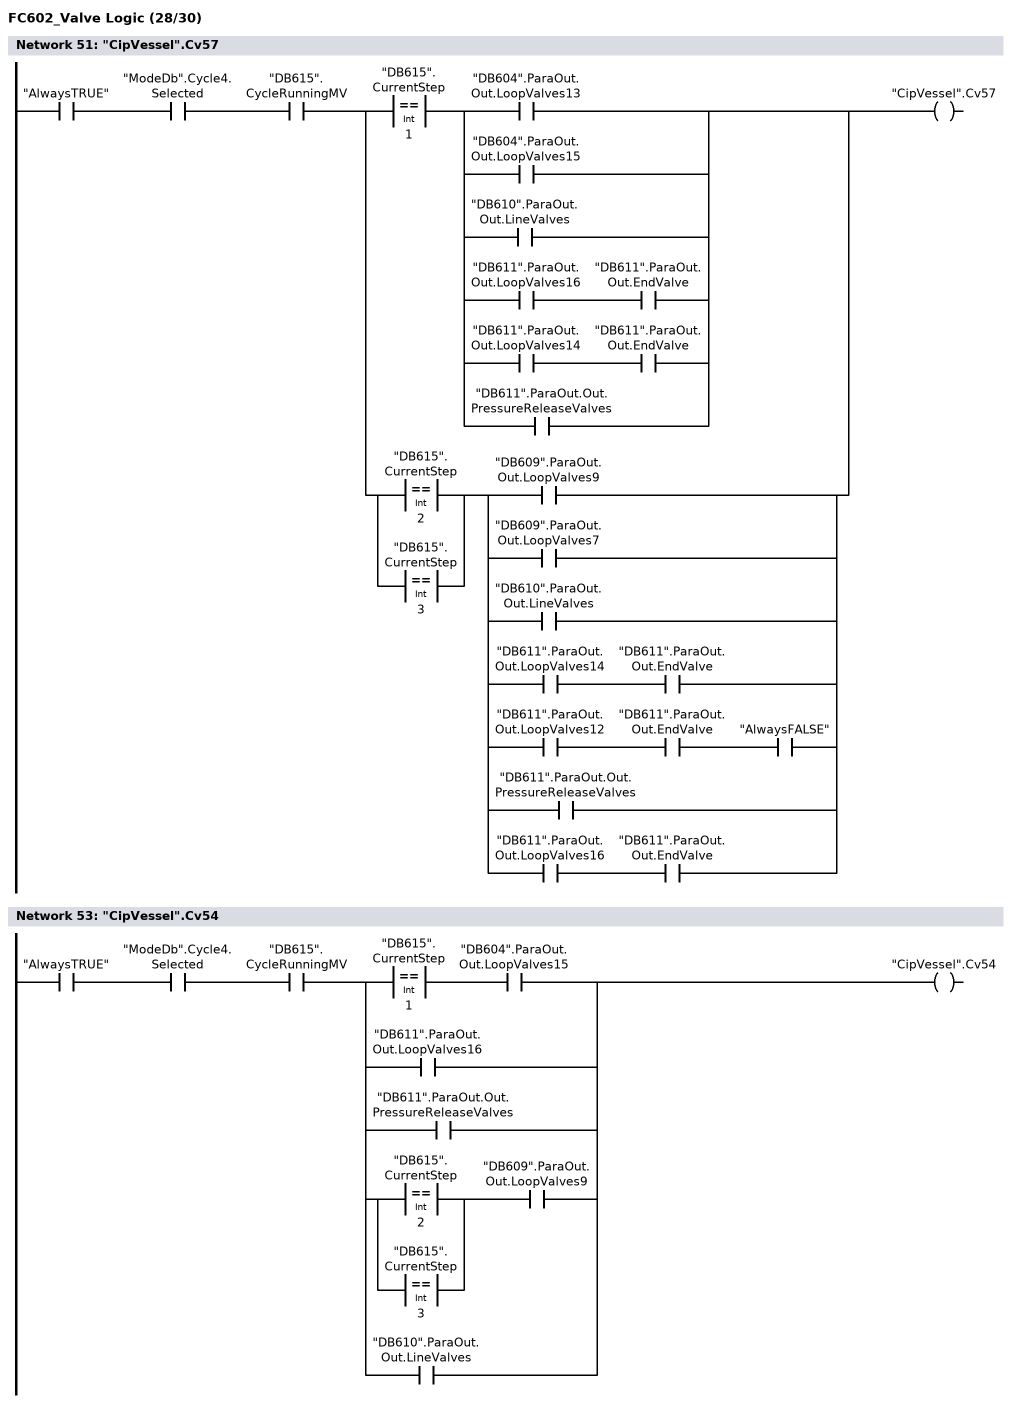
   RUNG wire#powerrail
      Contact( "AlwaysTRUE" )
      Contact( "ModeDb".Cycle4.Selected )
      Contact( "DB615".CycleRunningMV )
      wire#w1
      { S7_Templates := "SrcType := Int" } EQ_Contact(in1 := "DB615".CurrentStep, in2 := 1)
      wire#w2
      Contact( "DB604".ParaOut.Out.LoopValves13 )
      wire#w3
      Coil( "CipVessel".Cv57 )
   END_RUNG
   RUNG wire#w2
      Contact( "DB604".ParaOut.Out.LoopValves15 )
   END_RUNG wire#w3
   RUNG wire#w2
      Contact( "DB610".ParaOut.Out.LineValves )
   END_RUNG wire#w3
   RUNG wire#w2
      Contact( "DB611".ParaOut.Out.LoopValves16 )
      Contact( "DB611".ParaOut.Out.EndValve )
   END_RUNG wire#w3
   RUNG wire#w2
      Contact( "DB611".ParaOut.Out.LoopValves14 )
      Contact( "DB611".ParaOut.Out.EndValve )
   END_RUNG wire#w3
   RUNG wire#w2
      Contact( "DB611".ParaOut.Out.PressureReleaseValves )
   END_RUNG wire#w3
   RUNG wire#w1
      { S7_Templates := "SrcType := Int" } EQ_Contact(in1 := "DB615".CurrentStep, in2 := 2)
      wire#w4
      Contact( "DB609".ParaOut.Out.LoopValves9 )
   END_RUNG wire#w3
   RUNG wire#w1
      { S7_Templates := "SrcType := Int" } EQ_Contact(in1 := "DB615".CurrentStep, in2 := 3)
   END_RUNG wire#w4
   RUNG wire#w4
      Contact( "DB609".ParaOut.Out.LoopValves7 )
   END_RUNG wire#w3
   RUNG wire#w4
      Contact( "DB610".ParaOut.Out.LineValves )
   END_RUNG wire#w3
   RUNG wire#w4
      Contact( "DB611".ParaOut.Out.LoopValves14 )
      Contact( "DB611".ParaOut.Out.EndValve )
   END_RUNG wire#w3
   RUNG wire#w4
      Contact( "DB611".ParaOut.Out.LoopValves12 )
      Contact( "DB611".ParaOut.Out.EndValve )
      Contact( "AlwaysFALSE" )
   END_RUNG wire#w3
   RUNG wire#w4
      Contact( "DB611".ParaOut.Out.PressureReleaseValves )
   END_RUNG wire#w3
   RUNG wire#w4
      Contact( "DB611".ParaOut.Out.LoopValves16 )
      Contact( "DB611".ParaOut.Out.EndValve )
   END_RUNG wire#w3
   // the same network as SCL:
   "CipVessel".Cv57 := "AlwaysTRUE" AND "ModeDb".Cycle4.Selected AND "DB615".CycleRunningMV AND ((("DB615".CurrentStep = 1) AND ("DB604".ParaOut.Out.LoopValves13 OR "DB604".ParaOut.Out.LoopValves15 OR "DB610".ParaOut.Out.LineValves OR ("DB611".ParaOut.Out.LoopValves16 AND "DB611".ParaOut.Out.EndValve) OR ("DB611".ParaOut.Out.LoopValves14 AND "DB611".ParaOut.Out.EndValve) OR "DB611".ParaOut.Out.PressureReleaseValves)) OR ((("DB615".CurrentStep = 2) OR ("DB615".CurrentStep = 3)) AND ("DB609".ParaOut.Out.LoopValves9 OR "DB609".ParaOut.Out.LoopValves7 OR "DB610".ParaOut.Out.LineValves OR ("DB611".ParaOut.Out.LoopValves14 AND "DB611".ParaOut.Out.EndValve) OR ("DB611".ParaOut.Out.LoopValves12 AND "DB611".ParaOut.Out.EndValve AND "AlwaysFALSE") OR "DB611".ParaOut.Out.PressureReleaseValves OR ("DB611".ParaOut.Out.LoopValves16 AND "DB611".ParaOut.Out.EndValve))));
END_REGION

REGION Network 52: ---------- PTL LINE ------------
END_REGION

REGION Network 53: "CipVessel".Cv54
   RUNG wire#powerrail
      Contact( "AlwaysTRUE" )
      Contact( "ModeDb".Cycle4.Selected )
      Contact( "DB615".CycleRunningMV )
      wire#w1
      { S7_Templates := "SrcType := Int" } EQ_Contact(in1 := "DB615".CurrentStep, in2 := 1)
      Contact( "DB604".ParaOut.Out.LoopValves15 )
      wire#w2
      Coil( "CipVessel".Cv54 )
   END_RUNG
   RUNG wire#w1
      Contact( "DB611".ParaOut.Out.LoopValves16 )
   END_RUNG wire#w2
   RUNG wire#w1
      Contact( "DB611".ParaOut.Out.PressureReleaseValves )
   END_RUNG wire#w2
   RUNG wire#w1
      { S7_Templates := "SrcType := Int" } EQ_Contact(in1 := "DB615".CurrentStep, in2 := 2)
      wire#w3
      Contact( "DB609".ParaOut.Out.LoopValves9 )
   END_RUNG wire#w2
   RUNG wire#w1
      { S7_Templates := "SrcType := Int" } EQ_Contact(in1 := "DB615".CurrentStep, in2 := 3)
   END_RUNG wire#w3
   RUNG wire#w1
      Contact( "DB610".ParaOut.Out.LineValves )
   END_RUNG wire#w2
   // the same network as SCL:
   "CipVessel".Cv54 := "AlwaysTRUE" AND "ModeDb".Cycle4.Selected AND "DB615".CycleRunningMV AND ((("DB615".CurrentStep = 1) AND "DB604".ParaOut.Out.LoopValves15) OR "DB611".ParaOut.Out.LoopValves16 OR "DB611".ParaOut.Out.PressureReleaseValves OR ((("DB615".CurrentStep = 2) OR ("DB615".CurrentStep = 3)) AND "DB609".ParaOut.Out.LoopValves9) OR "DB610".ParaOut.Out.LineValves);
END_REGION

REGION Network 54: "CipVessel".Cv55
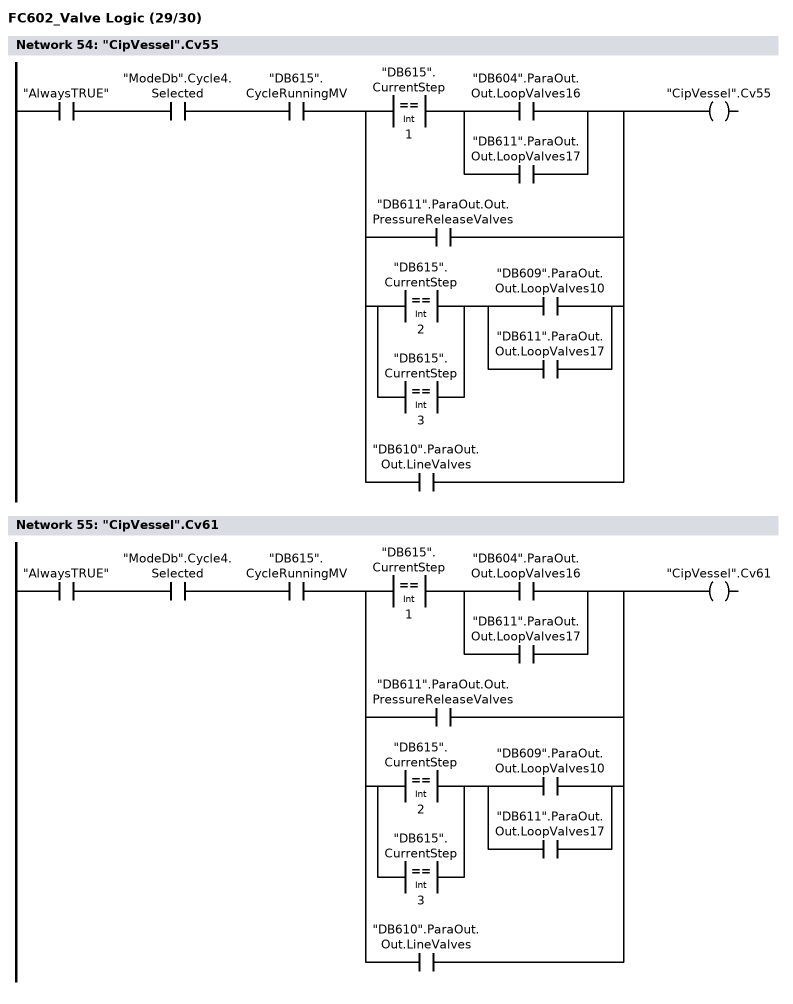
   RUNG wire#powerrail
      Contact( "AlwaysTRUE" )
      Contact( "ModeDb".Cycle4.Selected )
      Contact( "DB615".CycleRunningMV )
      wire#w1
      { S7_Templates := "SrcType := Int" } EQ_Contact(in1 := "DB615".CurrentStep, in2 := 1)
      wire#w2
      Contact( "DB604".ParaOut.Out.LoopValves16 )
      wire#w3
      Coil( "CipVessel".Cv55 )
   END_RUNG
   RUNG wire#w2
      Contact( "DB611".ParaOut.Out.LoopValves17 )
   END_RUNG wire#w3
   RUNG wire#w1
      Contact( "DB611".ParaOut.Out.PressureReleaseValves )
   END_RUNG wire#w3
   RUNG wire#w1
      { S7_Templates := "SrcType := Int" } EQ_Contact(in1 := "DB615".CurrentStep, in2 := 2)
      wire#w4
      Contact( "DB609".ParaOut.Out.LoopValves10 )
   END_RUNG wire#w3
   RUNG wire#w1
      { S7_Templates := "SrcType := Int" } EQ_Contact(in1 := "DB615".CurrentStep, in2 := 3)
   END_RUNG wire#w4
   RUNG wire#w4
      Contact( "DB611".ParaOut.Out.LoopValves17 )
   END_RUNG wire#w3
   RUNG wire#w1
      Contact( "DB610".ParaOut.Out.LineValves )
   END_RUNG wire#w3
   // the same network as SCL:
   "CipVessel".Cv55 := "AlwaysTRUE" AND "ModeDb".Cycle4.Selected AND "DB615".CycleRunningMV AND ((("DB615".CurrentStep = 1) AND ("DB604".ParaOut.Out.LoopValves16 OR "DB611".ParaOut.Out.LoopValves17)) OR "DB611".ParaOut.Out.PressureReleaseValves OR ((("DB615".CurrentStep = 2) OR ("DB615".CurrentStep = 3)) AND ("DB609".ParaOut.Out.LoopValves10 OR "DB611".ParaOut.Out.LoopValves17)) OR "DB610".ParaOut.Out.LineValves);
END_REGION

REGION Network 55: "CipVessel".Cv61
   RUNG wire#powerrail
      Contact( "AlwaysTRUE" )
      Contact( "ModeDb".Cycle4.Selected )
      Contact( "DB615".CycleRunningMV )
      wire#w1
      { S7_Templates := "SrcType := Int" } EQ_Contact(in1 := "DB615".CurrentStep, in2 := 1)
      wire#w2
      Contact( "DB604".ParaOut.Out.LoopValves16 )
      wire#w3
      Coil( "CipVessel".Cv61 )
   END_RUNG
   RUNG wire#w2
      Contact( "DB611".ParaOut.Out.LoopValves17 )
   END_RUNG wire#w3
   RUNG wire#w1
      Contact( "DB611".ParaOut.Out.PressureReleaseValves )
   END_RUNG wire#w3
   RUNG wire#w1
      { S7_Templates := "SrcType := Int" } EQ_Contact(in1 := "DB615".CurrentStep, in2 := 2)
      wire#w4
      Contact( "DB609".ParaOut.Out.LoopValves10 )
   END_RUNG wire#w3
   RUNG wire#w1
      { S7_Templates := "SrcType := Int" } EQ_Contact(in1 := "DB615".CurrentStep, in2 := 3)
   END_RUNG wire#w4
   RUNG wire#w4
      Contact( "DB611".ParaOut.Out.LoopValves17 )
   END_RUNG wire#w3
   RUNG wire#w1
      Contact( "DB610".ParaOut.Out.LineValves )
   END_RUNG wire#w3
   // the same network as SCL:
   "CipVessel".Cv61 := "AlwaysTRUE" AND "ModeDb".Cycle4.Selected AND "DB615".CycleRunningMV AND ((("DB615".CurrentStep = 1) AND ("DB604".ParaOut.Out.LoopValves16 OR "DB611".ParaOut.Out.LoopValves17)) OR "DB611".ParaOut.Out.PressureReleaseValves OR ((("DB615".CurrentStep = 2) OR ("DB615".CurrentStep = 3)) AND ("DB609".ParaOut.Out.LoopValves10 OR "DB611".ParaOut.Out.LoopValves17)) OR "DB610".ParaOut.Out.LineValves);
END_REGION

REGION Network 56: "CipVessel".Cv60
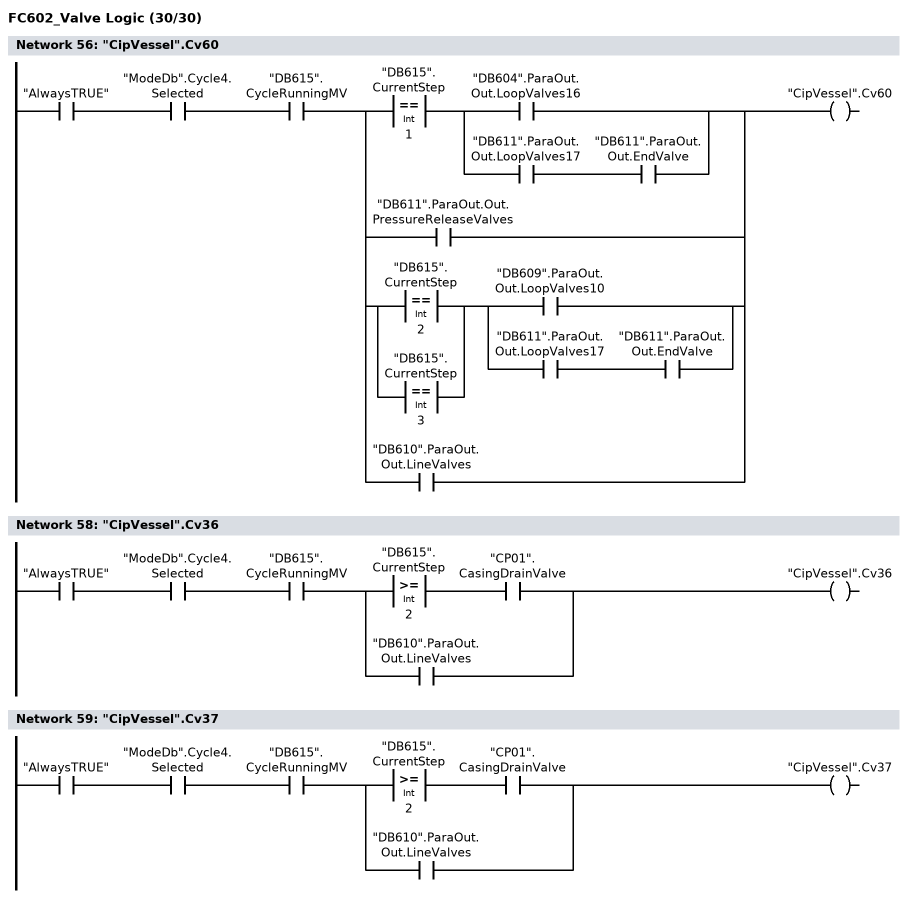
   RUNG wire#powerrail
      Contact( "AlwaysTRUE" )
      Contact( "ModeDb".Cycle4.Selected )
      Contact( "DB615".CycleRunningMV )
      wire#w1
      { S7_Templates := "SrcType := Int" } EQ_Contact(in1 := "DB615".CurrentStep, in2 := 1)
      wire#w2
      Contact( "DB604".ParaOut.Out.LoopValves16 )
      wire#w3
      Coil( "CipVessel".Cv60 )
   END_RUNG
   RUNG wire#w2
      Contact( "DB611".ParaOut.Out.LoopValves17 )
      Contact( "DB611".ParaOut.Out.EndValve )
   END_RUNG wire#w3
   RUNG wire#w1
      Contact( "DB611".ParaOut.Out.PressureReleaseValves )
   END_RUNG wire#w3
   RUNG wire#w1
      { S7_Templates := "SrcType := Int" } EQ_Contact(in1 := "DB615".CurrentStep, in2 := 2)
      wire#w4
      Contact( "DB609".ParaOut.Out.LoopValves10 )
   END_RUNG wire#w3
   RUNG wire#w1
      { S7_Templates := "SrcType := Int" } EQ_Contact(in1 := "DB615".CurrentStep, in2 := 3)
   END_RUNG wire#w4
   RUNG wire#w4
      Contact( "DB611".ParaOut.Out.LoopValves17 )
      Contact( "DB611".ParaOut.Out.EndValve )
   END_RUNG wire#w3
   RUNG wire#w1
      Contact( "DB610".ParaOut.Out.LineValves )
   END_RUNG wire#w3
   // the same network as SCL:
   "CipVessel".Cv60 := "AlwaysTRUE" AND "ModeDb".Cycle4.Selected AND "DB615".CycleRunningMV AND ((("DB615".CurrentStep = 1) AND ("DB604".ParaOut.Out.LoopValves16 OR ("DB611".ParaOut.Out.LoopValves17 AND "DB611".ParaOut.Out.EndValve))) OR "DB611".ParaOut.Out.PressureReleaseValves OR ((("DB615".CurrentStep = 2) OR ("DB615".CurrentStep = 3)) AND ("DB609".ParaOut.Out.LoopValves10 OR ("DB611".ParaOut.Out.LoopValves17 AND "DB611".ParaOut.Out.EndValve))) OR "DB610".ParaOut.Out.LineValves);
END_REGION

REGION Network 57: ----------PCD DRAIN------------
END_REGION

REGION Network 58: "CipVessel".Cv36
   RUNG wire#powerrail
      Contact( "AlwaysTRUE" )
      Contact( "ModeDb".Cycle4.Selected )
      Contact( "DB615".CycleRunningMV )
      wire#w1
      { S7_Templates := "SrcType := Int" } GE_Contact(in1 := "DB615".CurrentStep, in2 := 2)
      Contact( "CP01".CasingDrainValve )
      wire#w2
      Coil( "CipVessel".Cv36 )
   END_RUNG
   RUNG wire#w1
      Contact( "DB610".ParaOut.Out.LineValves )
   END_RUNG wire#w2
   // the same network as SCL:
   "CipVessel".Cv36 := "AlwaysTRUE" AND "ModeDb".Cycle4.Selected AND "DB615".CycleRunningMV AND ((("DB615".CurrentStep >= 2) AND "CP01".CasingDrainValve) OR "DB610".ParaOut.Out.LineValves);
END_REGION

REGION Network 59: "CipVessel".Cv37
   RUNG wire#powerrail
      Contact( "AlwaysTRUE" )
      Contact( "ModeDb".Cycle4.Selected )
      Contact( "DB615".CycleRunningMV )
      wire#w1
      { S7_Templates := "SrcType := Int" } GE_Contact(in1 := "DB615".CurrentStep, in2 := 2)
      Contact( "CP01".CasingDrainValve )
      wire#w2
      Coil( "CipVessel".Cv37 )
   END_RUNG
   RUNG wire#w1
      Contact( "DB610".ParaOut.Out.LineValves )
   END_RUNG wire#w2
   // the same network as SCL:
   "CipVessel".Cv37 := "AlwaysTRUE" AND "ModeDb".Cycle4.Selected AND "DB615".CycleRunningMV AND ((("DB615".CurrentStep >= 2) AND "CP01".CasingDrainValve) OR "DB610".ParaOut.Out.LineValves);
END_REGION
END_FUNCTION

FUNCTION "FC615" : Void
{ S7_Optimized_Access := 'TRUE' }
VERSION : 0.1

BEGIN
	REGION Common
	    IF "DB615".SelectStep = TRUE THEN
	        "DB615".TempStep := "DB615".CurrentStep;
	        REPEAT
	        "DB615".TempStep := "DB615".TempStep + 1;
	        UNTIL "DB623".StepEnable["DB615".TempStep] = TRUE OR ("DB615".TempStep > "DB616".TotalStep) END_REPEAT;
	        IF "DB615".TempStep <= "DB616".TotalStep THEN
	            "DB615".CurrentStep := "DB615".TempStep;
	        ELSE
	            "DB615".ProcessOver := 1;
	        END_IF;         
	        "DB615".SelectStep := false;
	    END_IF;
	    
	    
	    
	    IF "DB622".MainPopupMsg2 = 1 THEN
	        POKE_BLK(area_src := 16#84,
	                 dbNumber_src := 626,
	                 byteOffset_src := 0,
	                 area_dest := 16#84,
	                 dbNumber_dest := 625,
	                 byteOffset_dest := 0,
	                 count := 2382);  
	    END_IF;
	    
	END_REGION
	
	REGION common Set Para
	    "DB603".CycleSelection := "DB616".CycleSelection["DB615".CurrentStep];
	    
	    "DB604".ParaIn := "DB616".FillingInputPara["DB615".CurrentStep];
	    "DB607".SetTimeSecs := "DB616".MixingTimeInput["DB615".CurrentStep];
	    "DB608".ParaIn := "DB616".RecirculationInput["DB615".CurrentStep];
	    "DB609".ParaIn := "DB616".DrainInputs["DB615".CurrentStep];
	    "DB610".SetTime := "DB616".SystemDrainSetTimeInput["DB615".CurrentStep];
	    "DB611".ParaIn := "DB616".AirPurgingInputPara["DB615".CurrentStep];
	    "DB603".CycleSelection := "DB616".CycleSelection["DB615".CurrentStep];
	    
	    "DB609".ActualPressure := "AiDb".Ai11.ActValue;
	    "DB627".RepSv := "DB616".CycleSelection["DB615".CurrentStep].StepSelection.SetRepetition;
	    "DB627".RepPv := "DB603".ActualRepetition;
	    "DB604".ActualQuantity := "ModeDb".VesselWeight;
	    "DB609".ActualWeight := "ModeDb".VesselWeight;
	  //  "DB611".ActualPressure := "AiDb".Ai07.ActValue;
	    "DB609".ActualConductivityVessel := "AiDb".Ai15.ActValue;
	    "DB609".ParaIn.Parameters.SetConductivity := "DB623".FinalRinseSetCond;
	    "DB611".ActualPressure := "DB615".ApActPressure;
	    
	
	    "DB616".DrainInputs["DB615".CurrentStep].PreciseEngineering.DrainWeight := "DB624".VesselDrainWeight;
	    "DB616".DrainInputs["DB615".CurrentStep].Parameters.SetPressure := "DB623".DrainPressure;
	    "DB616".DrainInputs["DB615".CurrentStep].Parameters.PressureTolerance := "DB624".DrainPressureTolerance;
	    "DB616".DrainInputs["DB615".CurrentStep].ProductionSetting.CaiDelay := "CommonProductionSettings".CAIDelay;
	    
	    "DB616".SystemDrainSetTimeInput["DB615".CurrentStep] := "DB623".SystemDrainTime;
	    
	    "DB616".AirPurgingInputPara["DB615".CurrentStep].Parameters.SetPressure := "DB623".AirPurgingPressure;
	    "DB616".AirPurgingInputPara["DB615".CurrentStep].Parameters.PressureTolerance := "DB624".AirPurgingPressureTolerence;
	    "DB616".AirPurgingInputPara["DB615".CurrentStep].Parameters.VentOnTime := "DB624".AirPurgingReleaseTime;
	    "DB616".AirPurgingInputPara["DB615".CurrentStep].ProductionSetting.CAIDelay := "CommonProductionSettings".CAIDelay;
	    
	    
	    IF "DB611".StepDelay."Noof StepsPv" <= 1 THEN
	        "DB616".AirPurgingInputPara["DB615".CurrentStep].Selections.PressureMode := 0;
	    ELSE
	        "DB616".AirPurgingInputPara["DB615".CurrentStep].Selections.PressureMode := 1;
	    END_IF;
	    
	    "DB616".AirPurgingInputPara["DB615".CurrentStep].ProductionSetting.LoopDelay1 := "DB624".AirPurgeSamplingLineDelay;
	    "DB616".AirPurgingInputPara["DB615".CurrentStep].ProductionSetting.LoopDelay2 := "DB624".AirPurgeBlankeingLineDelay;
	    "DB616".AirPurgingInputPara["DB615".CurrentStep].ProductionSetting.LoopDelay3 := "DB624".AirPurgeJTubeLineDelay;
	    "DB616".AirPurgingInputPara["DB615".CurrentStep].ProductionSetting.LoopDelay4 := "DB624".AirPurgeSpargingLineDelay;
	    "DB616".AirPurgingInputPara["DB615".CurrentStep].ProductionSetting.LoopDelay5 := "DB624".AirPurgeSbiLineDelay;
	    "DB616".AirPurgingInputPara["DB615".CurrentStep].ProductionSetting.LoopDelay6 := "DB624".AirPurgeRecirculationlineDelay;
	    "DB616".AirPurgingInputPara["DB615".CurrentStep].ProductionSetting.LoopDelay7 := "DB624".AirPurgeVesselBypassLineDelay;
	    "DB616".AirPurgingInputPara["DB615".CurrentStep].ProductionSetting.LoopDelay8 := "DB624".AirPurgeVesselDrainLineDelay;
	    "DB616".AirPurgingInputPara["DB615".CurrentStep].ProductionSetting.LoopDelay9 := "DB624".AirPurgePumpBypassLineDelay;
	    "DB616".AirPurgingInputPara["DB615".CurrentStep].ProductionSetting.LoopDelay10 := "DB624".AirPurgePf01InLineDelay;
	    "DB616".AirPurgingInputPara["DB615".CurrentStep].ProductionSetting.LoopDelay11 := "DB624".AirPurgePf01VentLineDelay;
	    "DB616".AirPurgingInputPara["DB615".CurrentStep].ProductionSetting.LoopDelay12 := "DB624".AirPurgePf02InLineDelay;
	    "DB616".AirPurgingInputPara["DB615".CurrentStep].ProductionSetting.LoopDelay13 := "DB624".AirPurgePf02VentLineDelay;
	    "DB616".AirPurgingInputPara["DB615".CurrentStep].ProductionSetting.LoopDelay14 := "DB624".AirPurgePf02OutLineDelay;
	    "DB616".AirPurgingInputPara["DB615".CurrentStep].ProductionSetting.LoopDelay15 := "DB624".AirPurgePf01BypassLineDelay;
	    "DB616".AirPurgingInputPara["DB615".CurrentStep].ProductionSetting.LoopDelay16 := "DB624".AirPurgePf02BypassLineDelay;
	    "DB616".AirPurgingInputPara["DB615".CurrentStep].ProductionSetting.LoopDelay17 := "DB624".AirPurgePtlLineDelay;
	    
	END_REGION
	
	REGION Cycle 1 - PRE RINSE  CYCLE
	    
	    "DB616".CycleSelection[1].StepSelection.SetRepetition := "DB623".PreRinseCycleNoOfRep;
	    
	    "DB616".FillingInputPara[1].ProductionSetting.ZDVDelay := "CommonProductionSettings".WFIDelay;
	    "DB616".FillingInputPara[1].Parameters.PulsingOnTime := "DB623".SbiOnTime;
	    "DB616".FillingInputPara[1].Parameters.PulsingOffTime := "DB623".SbiOffTime;
	
	    "DB616".FillingInputPara[1].ProductionSetting.LoopDelay1 := "DB624".FillRinseSamplingLineDelay;
	    "DB616".FillingInputPara[1].ProductionSetting.LoopDelay2 := "DB624".FillRinseBlanketingLineDelay;
	    "DB616".FillingInputPara[1].ProductionSetting.LoopDelay3 := "DB624".FillRinseJTubeLineDelay;
	    "DB616".FillingInputPara[1].ProductionSetting.LoopDelay4 := "DB624".FillRinseSpargingLineDelay;
	    "DB616".FillingInputPara[1].ProductionSetting.LoopDelay5 := "DB624".FillRinseSbiLineDelay;
	    "DB616".FillingInputPara[1].ProductionSetting.LoopDelay6 := "DB624".FillRinseRecirculationlineDelay;
	    "DB616".FillingInputPara[1].ProductionSetting.LoopDelay7 := "DB624".FillRinseVesselBypassLineDelay;
	    "DB616".FillingInputPara[1].ProductionSetting.LoopDelay8 := "DB624".FillRinsePumpBypassLineDelay;
	    "DB616".FillingInputPara[1].ProductionSetting.LoopDelay9 := "DB624".FillRinsePf01InLineDelay;
	    "DB616".FillingInputPara[1].ProductionSetting.LoopDelay10 := "DB624".FillRinsePf01VentLineDelay;
	    "DB616".FillingInputPara[1].ProductionSetting.LoopDelay11 := "DB624".FillRinsePf02InLineDelay;
	    "DB616".FillingInputPara[1].ProductionSetting.LoopDelay12 := "DB624".FillRinsePf02VentLineDelay;
	    "DB616".FillingInputPara[1].ProductionSetting.LoopDelay13 := "DB624".FillRinsePf02OutLineDelay;
	    "DB616".FillingInputPara[1].ProductionSetting.LoopDelay14 := "DB624".FillRinsePf01BypassLineDelay;
	    "DB616".FillingInputPara[1].ProductionSetting.LoopDelay15 := "DB624".FillRinsePf02BypassLineDelay;
	    "DB616".FillingInputPara[1].ProductionSetting.LoopDelay16 := "DB624".FillRinsePtlLineDelay;
	    
	    
	    // "DB616".AirPurgingInputPara[1].ProductionSetting.LoopDelay1 := "DB624".AirPurgeSamplingLineDelay;
	    // "DB616".AirPurgingInputPara[1].ProductionSetting.LoopDelay2 := "DB624".AirPurgeBlankeingLineDelay;
	    // "DB616".AirPurgingInputPara[1].ProductionSetting.LoopDelay3 := "DB624".AirPurgeJTubeLineDelay;
	    // "DB616".AirPurgingInputPara[1].ProductionSetting.LoopDelay4 := "DB624".AirPurgeSpargingLineDelay;
	    // "DB616".AirPurgingInputPara[1].ProductionSetting.LoopDelay5 := "DB624".AirPurgeSbiLineDelay;
	    // "DB616".AirPurgingInputPara[1].ProductionSetting.LoopDelay6 := "DB624".AirPurgeRecirculationlineDelay;
	    // "DB616".AirPurgingInputPara[1].ProductionSetting.LoopDelay7 := "DB624".AirPurgeVesselBypassLineDelay;
	    // "DB616".AirPurgingInputPara[1].ProductionSetting.LoopDelay8 := "DB624".AirPurgeVesselDrainLineDelay ;
	    // "DB616".AirPurgingInputPara[1].ProductionSetting.LoopDelay9 := "DB624".AirPurgePumpBypassLineDelay ;
	    // "DB616".AirPurgingInputPara[1].ProductionSetting.LoopDelay10 := "DB624".AirPurgePf01InLineDelay ;
	    // "DB616".AirPurgingInputPara[1].ProductionSetting.LoopDelay11 := "DB624".AirPurgePf01VentLineDelay ;
	    // "DB616".AirPurgingInputPara[1].ProductionSetting.LoopDelay12 := "DB624".AirPurgePf02InLineDelay ;
	    // "DB616".AirPurgingInputPara[1].ProductionSetting.LoopDelay13 := "DB624".AirPurgePf02VentLineDelay ;
	    // "DB616".AirPurgingInputPara[1].ProductionSetting.LoopDelay14 := "DB624".AirPurgePf02OutLineDelay ;
	    // "DB616".AirPurgingInputPara[1].ProductionSetting.LoopDelay15 := "DB624".AirPurgePf01BypassLineDelay ;
	    // "DB616".AirPurgingInputPara[1].ProductionSetting.LoopDelay16 := "DB624".AirPurgePf02BypassLineDelay ;
	    // "DB616".AirPurgingInputPara[1].ProductionSetting.LoopDelay17 :="DB624".AirPurgePtlLineDelay ;
	    
	    // CASE "DB611".StepDelay."Noof StepsPv" OF
	    //     0..5:
	    //         "DB616".AirPurgingInputPara[1].Selections.PressureMode := 1;
	    //     6:
	    //         "DB616".AirPurgingInputPara[1].Selections.PressureMode := 0;
	    //     7..16:
	    //         "DB616".AirPurgingInputPara[1].Selections.PressureMode := 1;
	    //     ELSE
	    //         "DB616".AirPurgingInputPara[1].Selections.PressureMode := 1;
	    // END_CASE;
	            
	    
	    
	    REGION FILLING
	        IF "DB615".CurrentStep = 1 THEN
	            "DB616".FillingOutputPara[1] := "DB604".ParaOut;
	            "DB625".FillingPrint[1] := "DB604".Print;
	        ELSE
	            "DB616".FillingOutputPara[1] := "DB616".FillingOutputPara[0];
	        END_IF;
	    END_REGION
	    
	    REGION DRAIN
	        IF "DB615".CurrentStep = 1 AND "DB609".CycleEnable = 1 THEN
	            "DB616".DrainOutputs[1] := "DB609".ParaOut;
	
	        ELSE
	            "DB616".DrainOutputs[2] := "DB616".DrainOutputs[0];
	        END_IF;
	    END_REGION
	    
	    REGION SYSTEM DRAIN      
	        IF "DB615".CurrentStep = 1 THEN
	            "DB616".SystemDrainOutPara[1] := "DB610".ParaOut;
	        ELSE
	            "DB616".SystemDrainOutPara[1] := "DB616".SystemDrainOutPara[0];
	        END_IF;
	    END_REGION
	    
	    REGION AIR PURGE
	        IF "DB615".CurrentStep = 1 THEN
	            "DB616".AirPurgingOutPara[1] := "DB611".ParaOut;
	        ELSE
	            "DB616".AirPurgingOutPara[1] := "DB616".AirPurgingOutPara[0];
	        END_IF;
	    END_REGION
	    
	    REGION ON SCREEN PV
	        IF "DB615".CurrentStep = 1 THEN
	            //"DB627".FillQtySv := "DB623".Cyc1FillQty;
	            "DB627".FillQtyPv := "DB604".ActualQuantity;
	            //"DB627".TempSv := "DB623".Cyc1SetTemp;
	           // "DB627".TempPv := "DB605".ActualTemperature;
	            "DB627".MixingPv := "DB607".MixingTimer.TimeSecPV;
	            "DB627".MixingSv := "DB616".MixingTimeInput[1];
	        //    "DB627".APSv := "DB616".AirPurgingOutPara[1].Out.TimeSV;
	            "DB627".ApPv := "DB616".AirPurgingOutPara[1].Out.TimePV;
	            "DB627".APSv := "DB611".ParaOut.Out.TimeSV;
	            "DB627".ApReleaseTimeSv := "DB616".AirPurgingInputPara[1].Parameters.VentOnTime;
	            "DB627".ApReleaseTimePv := "DB616".AirPurgingOutPara[1].Out.PressureReleaseTimePV;
	            "DB627".SdSv := "DB623".SystemDrainTime;
	            "DB627".SdPv := "DB610".TimePv;
	           "DB627".RecirculationSv := "DB616".RecirculationOutput[1].Out.TimeSV;
	           "DB627".RecirculationPv := "DB616".RecirculationOutput[1].Out.TimePV;
	           "DB627".ConductivitySv := "DB609".ParaIn.Parameters.SetConductivity;
	           "DB627".ConductivityPv := "DB609".ActualConductivityVessel;
	         //   "DB627".DosingTimeSv := 0;
	         //   "DB627".DosingTimePv := 0;
	            "DB627".ApSetPressureSv := "DB623".AirPurgingPressure;
	            "DB627".ApSetPressurePv := "DB611".ActualPressure;
	            
	        END_IF;
	    END_REGION
	END_REGION
	
	REGION Cycle 2 - FILLING CYCLE
	    
	    "DB616".CycleSelection[2].StepSelection.SetRepetition := "DB623".FillingCycleNoOfRep;
	    
	    "DB616".FillingInputPara[2].ProductionSetting.ZDVDelay := "CommonProductionSettings".WFIDelay;
	   
	    "DB616".FillingInputPara[2].Parameters.FillQuantity1 := "DB623".FillingCycleFillQty;
	    
	    "DB616".FillingInputPara[2].ProductionSetting.LoopDelay1 := "DB624".FillRinseSamplingLineDelay;
	    "DB616".FillingInputPara[2].ProductionSetting.LoopDelay2 := "DB624".FillRinseBlanketingLineDelay;
	    "DB616".FillingInputPara[2].ProductionSetting.LoopDelay3 := "DB624".FillRinseJTubeLineDelay;
	    "DB616".FillingInputPara[2].ProductionSetting.LoopDelay4 := "DB624".FillRinseSpargingLineDelay;
	    
	    "DB616".MixingTimeInput[2] := "DB623".FillingCycleMixingTime;
	    
	    "DB616".RecirculationInput[2].Parameters.RecirculationInputToRunTime := "Cp01Cmd";
	    
	    "DB616".RecirculationInput[2].Parameters.LoopDelay1 := "DB624".RecSamplingLineDelay;
	    "DB616".RecirculationInput[2].Parameters.LoopDelay2 := "DB624".RecBlanketingLineDelay;
	    "DB616".RecirculationInput[2].Parameters.LoopDelay3 := "DB624".RecJTubeLineDelay;
	    "DB616".RecirculationInput[2].Parameters.LoopDelay4 := "DB624".RecSpargingLineDelay;
	    "DB616".RecirculationInput[2].Parameters.LoopDelay5 := "DB624".RecSbiLineDelay;
	    
	    IF "DB609".StepDelay."Noof StepsPv" <= 2 THEN
	        "DB616".DrainInputs[2].Selections.PressureModeSel := 1;
	        "DB616".DrainInputs[2].Selections.DrainPumpSel := 0;
	    ELSE
	        "DB616".DrainInputs[2].Selections.PressureModeSel := 0;
	        "DB616".DrainInputs[2].Selections.DrainPumpSel := 1;
	    END_IF;
	    
	    "DB616".DrainInputs[2].Selections.InputToRunPump := "DiFinal".Cp01FlowSwitch;
	    
	    "DB616".DrainInputs[2].ProductionSetting.LoopDelay1 := "DB624".DrainVesselDrainLineDelay;
	    "DB616".DrainInputs[2].ProductionSetting.LoopDelay2 := "DB624".DrainPumpBypassLineDelay;
	    "DB616".DrainInputs[2].ProductionSetting.LoopDelay3 := "DB624".DrainPf01InLineDelay;
	    "DB616".DrainInputs[2].ProductionSetting.LoopDelay4 := "DB624".DrainPf01VentLineDelay;
	    "DB616".DrainInputs[2].ProductionSetting.LoopDelay5 := "DB624".DrainPf02InLineDelay;
	    "DB616".DrainInputs[2].ProductionSetting.LoopDelay6 :="DB624".DrainPf02VentLineDelay ;
	    "DB616".DrainInputs[2].ProductionSetting.LoopDelay7 :="DB624".DrainPf02OutLineDelay ;
	    "DB616".DrainInputs[2].ProductionSetting.LoopDelay8 :="DB624".DrainPf01BypassLineDelay ;
	    "DB616".DrainInputs[2].ProductionSetting.LoopDelay9 :="DB624".DrainPf02BypassLineDelay ;
	    
	    // IF "DB611".StepDelay."Noof StepsPv" = 1 THEN
	    //     "DB616".AirPurgingInputPara[2].Selections.PressureMode := 0;
	    // ELSE
	    //     "DB616".AirPurgingInputPara[2].Selections.PressureMode := 1;
	    // END_IF;
	    
	    // "DB616".AirPurgingInputPara[2].ProductionSetting.LoopDelay1 := "DB624".AirPurgeSamplingLineDelay;
	    // "DB616".AirPurgingInputPara[2].ProductionSetting.LoopDelay2 := "DB624".AirPurgeBlankeingLineDelay;
	    // "DB616".AirPurgingInputPara[2].ProductionSetting.LoopDelay3 := "DB624".AirPurgeJTubeLineDelay;
	    // "DB616".AirPurgingInputPara[2].ProductionSetting.LoopDelay4 := "DB624".AirPurgeSpargingLineDelay;
	    // "DB616".AirPurgingInputPara[2].ProductionSetting.LoopDelay5 := "DB624".AirPurgeSbiLineDelay;
	    // "DB616".AirPurgingInputPara[2].ProductionSetting.LoopDelay6 := "DB624".AirPurgeVesselDrainLineDelay;
	    // "DB616".AirPurgingInputPara[2].ProductionSetting.LoopDelay7 := "DB624".AirPurgePumpBypassLineDelay;
	    // "DB616".AirPurgingInputPara[2].ProductionSetting.LoopDelay8 := "DB624".AirPurgePf01InLineDelay;
	    // "DB616".AirPurgingInputPara[2].ProductionSetting.LoopDelay9 := "DB624".AirPurgePf01VentLineDelay;
	    // "DB616".AirPurgingInputPara[2].ProductionSetting.LoopDelay10 := "DB624".AirPurgePf02InLineDelay;
	    // "DB616".AirPurgingInputPara[2].ProductionSetting.LoopDelay11 := "DB624".AirPurgePf02VentLineDelay;
	    // "DB616".AirPurgingInputPara[2].ProductionSetting.LoopDelay12 := "DB624".AirPurgePf02OutLineDelay;
	    // "DB616".AirPurgingInputPara[2].ProductionSetting.LoopDelay13 := "DB624".AirPurgePf01BypassLineDelay;
	    // "DB616".AirPurgingInputPara[2].ProductionSetting.LoopDelay14 := "DB624".AirPurgePf02BypassLineDelay;
	    // "DB616".AirPurgingInputPara[2].ProductionSetting.LoopDelay15 := "DB624".AirPurgePtlLineDelay;
	    
	    REGION FILLING
	        IF "DB615".CurrentStep = 2 THEN
	            "DB616".FillingOutputPara[2] := "DB604".ParaOut;
	            "DB625".FillingPrint[2] := "DB604".Print;
	        ELSE
	            "DB616".FillingOutputPara[2] := "DB616".FillingOutputPara[0];
	        END_IF;
	    END_REGION
	   
	    REGION MIXING
	        IF "DB615".CurrentStep = 2 AND "DB607".CycleEnable = 1 THEN
	            "DB625".MixingTime[2] := "DB607".Print;
	        END_IF;
	    END_REGION
	    
	    REGION RECIRCULATION
	        IF "DB615".CurrentStep = 2 THEN
	            "DB616".RecirculationOutput[2] := "DB608".ParaOut;
	            //"DB625".RecirculationPrint[2] := "DB608".Print;
	        ELSE
	            "DB616".RecirculationOutput[2] := "DB616".RecirculationOutput[0];
	        END_IF;
	    END_REGION
	    
	    REGION DRAIN
	        IF "DB615".CurrentStep = 2 AND "DB609".CycleEnable = 1 THEN
	            "DB616".DrainOutputs[2] := "DB609".ParaOut;
	
	        ELSE
	            "DB616".DrainOutputs[2] := "DB616".DrainOutputs[0];
	        END_IF;
	    END_REGION
	    
	    REGION SYSTEM DRAIN      
	        IF "DB615".CurrentStep = 2 THEN
	            "DB616".SystemDrainOutPara[2] := "DB610".ParaOut;
	        ELSE
	            "DB616".SystemDrainOutPara[2] := "DB616".SystemDrainOutPara[0];
	        END_IF;
	    END_REGION
	    
	    REGION AIR PURGE
	        IF "DB615".CurrentStep = 2 THEN
	            "DB616".AirPurgingOutPara[2] := "DB611".ParaOut;
	        ELSE
	            "DB616".AirPurgingOutPara[2] := "DB616".AirPurgingOutPara[0];
	        END_IF;
	    END_REGION
	    
	    REGION ON SCREEN PV
	        IF "DB615".CurrentStep = 2 THEN
	            "DB627".RinseTimeSv := 0;
	            "DB627".RinseTimePv := 0;
	            "DB627".RepSv :=  "DB623".FillingCycleNoOfRep;
	            "DB627".RepPv := "DB603".ActualRepetition;
	            "DB627".SdSv := "DB623".SystemDrainTime;
	            "DB627".SdPv := "DB610".Timer.TimeSecPV;
	            "DB627".MixingSv := "DB616".MixingTimeInput[2] ;
	            "DB627".MixingPv := "DB607".MixingTimer.TimeSecPV;
	            //"DB627".FillQtySv :=  "DB616".FillingInputPara[2].Parameters.FillQuantity1;
	            "DB627".FillQtyPv :=  "ModeDb".VesselWeight;
	            "DB627".ApReleaseTimeSv := "DB624".AirPurgingReleaseTime;
	            "DB627".ApReleaseTimePv := "DB611".ParaOut.Out.PressureReleaseTimePV;
	            "DB627".FillQtySv := "DB623".FillingCycleFillQty;
	          //  "DB627".FillQtyPv := "DB604".ActualQuantity;
	            //"DB627".TempSv := "DB623".Cyc1SetTemp;
	            // "DB627".TempPv := "DB605".ActualTemperature;
	        //    "DB627".APSv := "DB616".AirPurgingOutPara[2].Out.TimeSV;
	            "DB627".ApPv := "DB616".AirPurgingOutPara[2].Out.TimePV;
	            "DB627".APSv := "DB611".ParaOut.Out.TimeSV;
	          //  "DB627".RecirculationSv := "DB616".RecirculationOutput[2].Out.TimeSV;
	            "DB627".RecirculationPv := "DB616".RecirculationOutput[2].Out.TimePV;
	            "DB627".RecirculationSv := "DB608".ParaOut.Out.TimeSV;
	            "DB627".ConductivitySv := "DB609".ParaIn.Parameters.SetConductivity;
	            "DB627".ConductivityPv := "DB609".ActualConductivityVessel;
	            //   "DB627".DosingTimeSv := 0;
	            //   "DB627".DosingTimePv := 0;
	            "DB627".ApSetPressureSv := "DB623".AirPurgingPressure;
	            "DB627".ApSetPressurePv := "DB611".ActualPressure;
	            
	        END_IF;
	    END_REGION
	END_REGION
	
	REGION Cycle 3 - FINAL RINSE CYCLE
	    
	    "DB616".CycleSelection[3].StepSelection.SetRepetition := "DB624"."FinalRinseCycleNo.OfRep";
	    
	    "DB616".FillingInputPara[3].ProductionSetting.ZDVDelay := "CommonProductionSettings".WFIDelay;
	    
	    "DB616".FillingInputPara[3].Parameters.FillQuantity1 := "DB623".FinalRinseCycleFillQty;
	    
	    "DB616".FillingInputPara[3].ProductionSetting.LoopDelay1 := "DB624".FillRinseSamplingLineDelay;
	    "DB616".FillingInputPara[3].ProductionSetting.LoopDelay2 := "DB624".FillRinseBlanketingLineDelay;
	    "DB616".FillingInputPara[3].ProductionSetting.LoopDelay3 := "DB624".FillRinseJTubeLineDelay;
	    "DB616".FillingInputPara[3].ProductionSetting.LoopDelay4 := "DB624".FillRinseSpargingLineDelay;
	    
	    "DB616".MixingTimeInput[3] := "DB623".FinalRinseCycleMixingTime;
	    
	    "DB616".RecirculationInput[3].Parameters.RecirculationInputToRunTime := "Cp01Cmd";
	    "DB616".RecirculationInput[3].Parameters.LoopDelay1 := "DB624".RecSamplingLineDelay;
	    "DB616".RecirculationInput[3].Parameters.LoopDelay2 := "DB624".RecBlanketingLineDelay;
	    "DB616".RecirculationInput[3].Parameters.LoopDelay3 := "DB624".RecJTubeLineDelay;
	    "DB616".RecirculationInput[3].Parameters.LoopDelay4 := "DB624".RecSpargingLineDelay;
	    "DB616".RecirculationInput[3].Parameters.LoopDelay5 := "DB624".RecSbiLineDelay;
	    
	    //"DB616".DrainInputs[3].ProductionSetting.LoopDelay1 := "DB624".FinalRinseCycleVesselDrainLineDelay;
	    "DB616".DrainInputs[3].ProductionSetting.DelayToCheckConductivity := "DB624".DelayToCheckConductivity;
	    "DB616".DrainInputs[3].ProductionSetting.ConductivityCheckTime := "DB624".ConductivityCheckTime;
	    
	    IF "DB609".StepDelay."Noof StepsPv" <= 2 THEN
	        "DB616".DrainInputs[3].Selections.PressureModeSel := 1;
	        "DB616".DrainInputs[3].Selections.DrainPumpSel := 0;
	    ELSE
	        "DB616".DrainInputs[3].Selections.PressureModeSel := 0;
	        "DB616".DrainInputs[3].Selections.DrainPumpSel := 1;
	    END_IF;
	    
	    "DB616".DrainInputs[3].Selections.InputToRunPump := "DiFinal".Cp01FlowSwitch;
	    
	    "DB616".DrainInputs[3].ProductionSetting.LoopDelay1 := "DB624".DrainVesselDrainLineDelay;
	    "DB616".DrainInputs[3].ProductionSetting.LoopDelay2 := "DB624".DrainPumpBypassLineDelay;
	    "DB616".DrainInputs[3].ProductionSetting.LoopDelay3 := "DB624".DrainPf01InLineDelay;
	    "DB616".DrainInputs[3].ProductionSetting.LoopDelay4 := "DB624".DrainPf01VentLineDelay;
	    "DB616".DrainInputs[3].ProductionSetting.LoopDelay5 := "DB624".DrainPf02InLineDelay;
	    "DB616".DrainInputs[3].ProductionSetting.LoopDelay6 := "DB624".DrainPf02VentLineDelay;
	    "DB616".DrainInputs[3].ProductionSetting.LoopDelay7 := "DB624".DrainPf02OutLineDelay;
	    "DB616".DrainInputs[3].ProductionSetting.LoopDelay8 := "DB624".DrainPf01BypassLineDelay;
	    "DB616".DrainInputs[3].ProductionSetting.LoopDelay9 := "DB624".DrainPf02BypassLineDelay;
	    
	    // "DB616".AirPurgingInputPara[2].ProductionSetting.LoopDelay1 := "DB624".AirPurgeSamplingLineDelay;
	    // "DB616".AirPurgingInputPara[2].ProductionSetting.LoopDelay2 := "DB624".AirPurgeBlankeingLineDelay;
	    // "DB616".AirPurgingInputPara[2].ProductionSetting.LoopDelay3 := "DB624".AirPurgeJTubeLineDelay;
	    // "DB616".AirPurgingInputPara[2].ProductionSetting.LoopDelay4 := "DB624".AirPurgeSpargingLineDelay;
	    // "DB616".AirPurgingInputPara[2].ProductionSetting.LoopDelay5 := "DB624".AirPurgeSbiLineDelay;
	    // "DB616".AirPurgingInputPara[2].ProductionSetting.LoopDelay6 := "DB624".AirPurgeVesselDrainLineDelay;
	    
	END_REGION
	REGION FILLING
	    IF "DB615".CurrentStep = 3 THEN
	        "DB616".FillingOutputPara[3] := "DB604".ParaOut;
	        "DB625".FillingPrint[3] := "DB604".Print;
	    ELSE
	        "DB616".FillingOutputPara[3] := "DB616".FillingOutputPara[0];
	    END_IF;
	END_REGION
	
	REGION MIXING
	    IF "DB615".CurrentStep = 3 AND "DB607".CycleEnable = 1 THEN
	        "DB625".MixingTime[3] := "DB607".Print;
	    END_IF;
	END_REGION
	
	REGION RECIRCULATION
	    IF "DB615".CurrentStep = 3 THEN
	        "DB616".RecirculationOutput[3] := "DB608".ParaOut;
	        //"DB625".RecirculationPrint[2] := "DB608".Print;
	    ELSE
	        "DB616".RecirculationOutput[3] := "DB616".RecirculationOutput[0];
	    END_IF;
	END_REGION
	
	REGION DRAIN
	    IF "DB615".CurrentStep = 3 AND "DB609".CycleEnable = 1 THEN
	        "DB616".DrainOutputs[3] := "DB609".ParaOut;
	        
	    ELSE
	        "DB616".DrainOutputs[3] := "DB616".DrainOutputs[0];
	    END_IF;
	END_REGION
	
	REGION SYSTEM DRAIN      
	    IF "DB615".CurrentStep = 3 THEN
	        "DB616".SystemDrainOutPara[3] := "DB610".ParaOut;
	    ELSE
	        "DB616".SystemDrainOutPara[3] := "DB616".SystemDrainOutPara[0];
	    END_IF;
	END_REGION
	
	REGION AIR PURGE
	    IF "DB615".CurrentStep = 3 THEN
	        "DB616".AirPurgingOutPara[3] := "DB611".ParaOut;
	    ELSE
	        "DB616".AirPurgingOutPara[3] := "DB616".AirPurgingOutPara[0];
	    END_IF;
	END_REGION
	REGION ON SCREEN PV
	    IF "DB615".CurrentStep = 3 THEN
	        "DB627".RinseTimeSv := 0;
	        "DB627".RinseTimePv := 0;
	        "DB627".RepSv := "DB623".FillingCycleNoOfRep;
	        "DB627".RepPv := "DB603".ActualRepetition;
	        "DB627".SdSv := "DB623".SystemDrainTime;
	        "DB627".SdPv := "DB610".Timer.TimeSecPV;
	        "DB627".MixingSv := "DB616".MixingTimeInput[3];
	        "DB627".MixingPv := "DB607".MixingTimer.TimeSecPV;
	        //"DB627".FillQtySv :=  "DB616".FillingInputPara[2].Parameters.FillQuantity1;
	        "DB627".FillQtyPv := "ModeDb".VesselWeight;
	        "DB627".ApReleaseTimeSv := "DB624".AirPurgingReleaseTime;
	        "DB627".ApReleaseTimePv := "DB611".ParaOut.Out.PressureReleaseTimePV;
	        "DB627".FillQtySv := "DB623".FinalRinseCycleFillQty;
	        //  "DB627".FillQtyPv := "DB604".ActualQuantity;
	        //"DB627".TempSv := "DB623".Cyc1SetTemp;
	        // "DB627".TempPv := "DB605".ActualTemperature;
	      //  "DB627".APSv := "DB616".AirPurgingOutPara[2].Out.TimeSV;
	        "DB627".ApPv := "DB616".AirPurgingOutPara[3].Out.TimePV;
	        "DB627".APSv := "DB611".ParaOut.Out.TimeSV;
	      //  "DB627".RecirculationSv := "DB616".RecirculationOutput[2].Out.TimeSV;
	        "DB627".RecirculationPv := "DB616".RecirculationOutput[3].Out.TimePV;
	        "DB627".RecirculationSv := "DB608".ParaOut.Out.TimeSV;
	        "DB627".ConductivitySv := "DB609".ParaIn.Parameters.SetConductivity;
	        "DB627".ConductivityPv := "DB609".ActualConductivityVessel;
	        //   "DB627".DosingTimeSv := 0;
	        //   "DB627".DosingTimePv := 0;
	        "DB627".ApSetPressureSv := "DB623".AirPurgingPressure;
	        "DB627".ApSetPressurePv := "DB611".ActualPressure;
	        
	    END_IF;
	END_REGION
	
	
	
	
END_FUNCTION

FUNCTION_BLOCK "FB614"   // FB614, LAD
TITLE = FB614
{ S7_Optimized_Access := 'TRUE' }
// CIP FSC PUMP
// stored: AutoNumber false, MemoryReserve 100, SetENOAutomatically false
   VAR_INPUT
      Simulation : Bool;
      Running : Bool;
      OnCondition : Bool;
      FscInput : Bool;
      BypassFscLogic : Bool;
      OnDelay : Int;
      OffDelay : Int;
      CasingDrainDelay : Int;
   END_VAR
   VAR_OUTPUT
      Output : Bool;
      CasingDrainValve : Bool;
   END_VAR
   VAR_IN_OUT
      Temp1 : DInt;
      Temp2 : DInt;
      Temp3 : Bool;
      Temp4 : Bool;
      Temp5 : DInt;
   END_VAR
   VAR
      OnDelayTimer { S7_SetPoint := 'True'} : TON_TIME;
      BypassFSLogicForcefully { S7_SetPoint := 'True'} : TON_TIME;
      OffDelayTimer { S7_SetPoint := 'True'} : TON_TIME;
      CdTimer { S7_SetPoint := 'True'} : TON_TIME;
   END_VAR
   VAR_TEMP   // added for the SCL form of the ladder/FBD networks
      _w1 : Bool;
   END_VAR
BEGIN

REGION Network 1
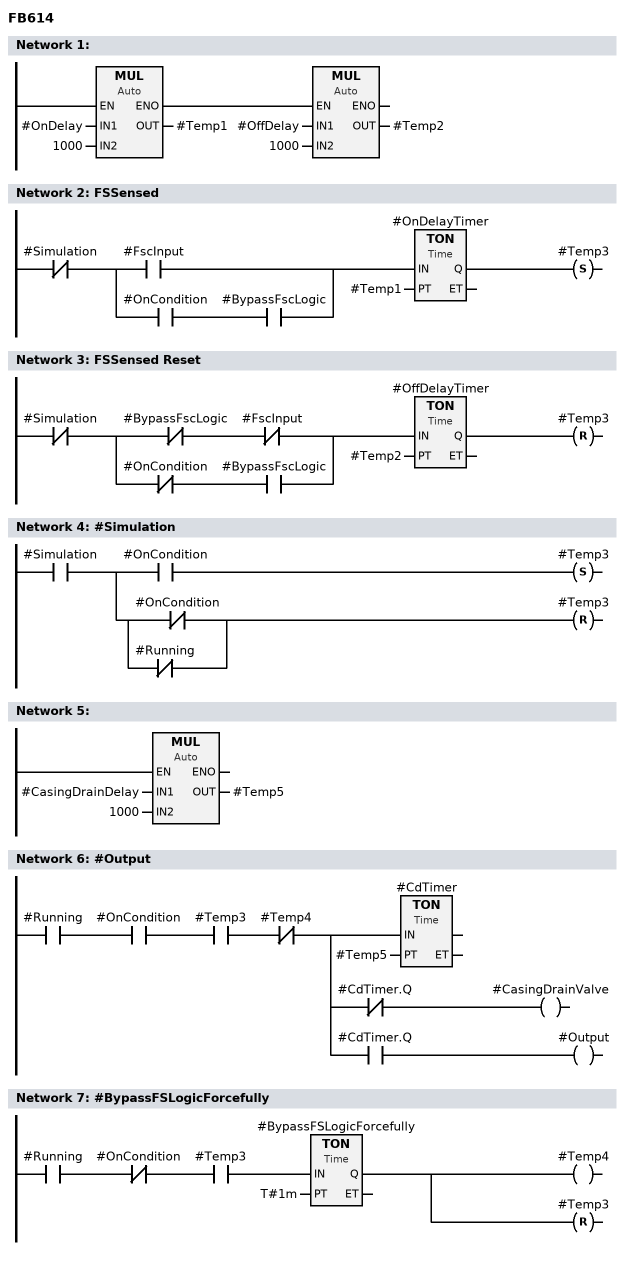
   RUNG wire#powerrail
      Mul(in1 := #OnDelay, in2 := 1000, out => #Temp1)
      Mul(in1 := #OffDelay, in2 := 1000, out => #Temp2)
   END_RUNG
   // the same network as SCL:
   #Temp1 := #OnDelay * 1000;
   #Temp2 := #OffDelay * 1000;
END_REGION

REGION Network 2: FSSensed
   RUNG wire#powerrail
      I_Contact( #Simulation )
      wire#w1
      Contact( #FscInput )
      wire#w2
      { S7_Templates := "time_type := Time" } #OnDelayTimer.TON(pt := #Temp1, et =>)
      S_Coil( #Temp3 )
   END_RUNG
   RUNG wire#w1
      Contact( #OnCondition )
      Contact( #BypassFscLogic )
   END_RUNG wire#w2
   // the same network as SCL:
   #OnDelayTimer(IN := NOT #Simulation AND (#FscInput OR (#OnCondition AND #BypassFscLogic)), PT := #Temp1);   // TON
   IF #OnDelayTimer.Q THEN #Temp3 := TRUE; END_IF;
END_REGION

REGION Network 3: FSSensed Reset
   RUNG wire#powerrail
      I_Contact( #Simulation )
      wire#w1
      I_Contact( #BypassFscLogic )
      I_Contact( #FscInput )
      wire#w2
      { S7_Templates := "time_type := Time" } #OffDelayTimer.TON(pt := #Temp2, et =>)
      R_Coil( #Temp3 )
   END_RUNG
   RUNG wire#w1
      I_Contact( #OnCondition )
      Contact( #BypassFscLogic )
   END_RUNG wire#w2
   // the same network as SCL:
   #OffDelayTimer(IN := NOT #Simulation AND ((NOT #BypassFscLogic AND NOT #FscInput) OR (NOT #OnCondition AND #BypassFscLogic)),   // TON
                  PT := #Temp2);
   IF #OffDelayTimer.Q THEN #Temp3 := FALSE; END_IF;
END_REGION

REGION Network 4: #Simulation
   RUNG wire#powerrail
      Contact( #Simulation )
      wire#w1
      Contact( #OnCondition )
      S_Coil( #Temp3 )
   END_RUNG
   RUNG wire#w1
      I_Contact( #OnCondition )
      wire#w2
      R_Coil( #Temp3 )
   END_RUNG
   RUNG wire#w1
      I_Contact( #Running )
   END_RUNG wire#w2
   // the same network as SCL:
   IF #Simulation AND #OnCondition THEN #Temp3 := TRUE; END_IF;
   IF #Simulation AND (NOT #OnCondition OR NOT #Running) THEN #Temp3 := FALSE; END_IF;
END_REGION

REGION Network 5
   RUNG wire#powerrail
      Mul(in1 := #CasingDrainDelay, in2 := 1000, out => #Temp5)
   END_RUNG
   // the same network as SCL:
   #Temp5 := #CasingDrainDelay * 1000;
END_REGION

REGION Network 6: #Output
   RUNG wire#powerrail
      Contact( #Running )
      Contact( #OnCondition )
      Contact( #Temp3 )
      I_Contact( #Temp4 )
      wire#w1
      { S7_Templates := "time_type := Time" } #CdTimer.TON(pt := #Temp5, et =>)
   END_RUNG
   RUNG wire#w1
      I_Contact( #CdTimer.Q )
      Coil( #CasingDrainValve )
   END_RUNG
   RUNG wire#w1
      Contact( #CdTimer.Q )
      Coil( #Output )
   END_RUNG
   // the same network as SCL:
   #_w1 := #Running AND #OnCondition AND #Temp3 AND NOT #Temp4;
   #CdTimer(IN := #_w1, PT := #Temp5);   // TON
   #CasingDrainValve := #_w1 AND NOT #CdTimer.Q;
   #Output := #_w1 AND #CdTimer.Q;
END_REGION

REGION Network 7: #BypassFSLogicForcefully
   RUNG wire#powerrail
      Contact( #Running )
      I_Contact( #OnCondition )
      Contact( #Temp3 )
      { S7_Templates := "time_type := Time" } #BypassFSLogicForcefully.TON(pt := T#1m, et =>)
      wire#w1
      Coil( #Temp4 )
   END_RUNG
   RUNG wire#w1
      R_Coil( #Temp3 )
   END_RUNG
   // the same network as SCL:
   #BypassFSLogicForcefully(IN := #Running AND NOT #OnCondition AND #Temp3, PT := T#1m);   // TON
   #Temp4 := #BypassFSLogicForcefully.Q;
   IF #BypassFSLogicForcefully.Q THEN #Temp3 := FALSE; END_IF;
END_REGION
END_FUNCTION_BLOCK

FUNCTION "PidInitialisation" : Void   // FC3, LAD
{ S7_Optimized_Access := 'TRUE' }
// stored: SetENOAutomatically false
BEGIN

REGION Network 2: CV30 Parameters SIP
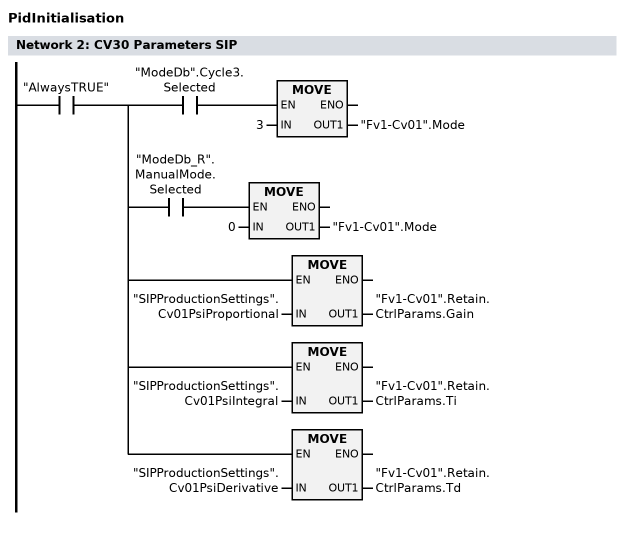
   RUNG wire#powerrail
      Contact( "AlwaysTRUE" )
      wire#w1
      Contact( "ModeDb".Cycle3.Selected )
      { S7_GenerateENO := "TRUE" } Move(in := 3, out1 => "Fv1-Cv01".Mode)
   END_RUNG
   RUNG wire#w1
      Contact( "ModeDb_R".ManualMode.Selected )
      { S7_GenerateENO := "TRUE" } Move(in := 0, out1 => "Fv1-Cv01".Mode)
   END_RUNG
   RUNG wire#w1
      { S7_GenerateENO := "TRUE" } Move(in := "SIPProductionSettings".Cv01PsiProportional, out1 => "Fv1-Cv01".Retain.CtrlParams.Gain)
   END_RUNG
   RUNG wire#w1
      { S7_GenerateENO := "TRUE" } Move(in := "SIPProductionSettings".Cv01PsiIntegral, out1 => "Fv1-Cv01".Retain.CtrlParams.Ti)
   END_RUNG
   RUNG wire#w1
      { S7_GenerateENO := "TRUE" } Move(in := "SIPProductionSettings".Cv01PsiDerivative, out1 => "Fv1-Cv01".Retain.CtrlParams.Td)
   END_RUNG
   // the same network as SCL:
   IF "AlwaysTRUE" AND "ModeDb".Cycle3.Selected THEN "Fv1-Cv01".Mode := 3; END_IF;
   IF "AlwaysTRUE" AND "ModeDb_R".ManualMode.Selected THEN "Fv1-Cv01".Mode := 0; END_IF;
   IF "AlwaysTRUE" THEN
       "Fv1-Cv01".Retain.CtrlParams.Gain := "SIPProductionSettings".Cv01PsiProportional;
       "Fv1-Cv01".Retain.CtrlParams.Ti := "SIPProductionSettings".Cv01PsiIntegral;
       "Fv1-Cv01".Retain.CtrlParams.Td := "SIPProductionSettings".Cv01PsiDerivative;
   END_IF;
END_REGION
END_FUNCTION

ORGANIZATION_BLOCK "Startup"   // OB100, LAD, Startup
TITLE = "Complete Restart"
{ S7_Optimized_Access := 'TRUE' }
// stored: AutoNumber false, SetENOAutomatically false
   VAR_INPUT
      LostRetentive : Bool;   // True if retentive data are lost
      LostRTC : Bool;   // True if date and time are lost
   END_VAR
BEGIN

REGION Network 1
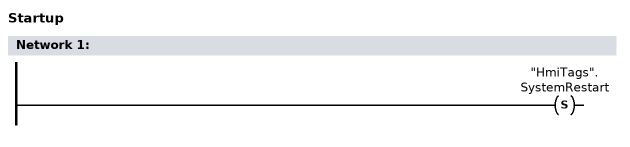
   RUNG wire#powerrail
      S_Coil( "HmiTags".SystemRestart )
   END_RUNG
   // the same network as SCL:
   "HmiTags".SystemRestart := TRUE;
END_REGION
END_ORGANIZATION_BLOCK

ORGANIZATION_BLOCK "Date_Time_Block"   // OB200, LAD, ProgramCycle
{ S7_Optimized_Access := 'TRUE' }
// stored: SetENOAutomatically false
   VAR_TEMP   // added for the SCL form of the ladder/FBD networks
      _w1 : Bool;
      _w2 : Bool;
      _w3 : Bool;
   END_VAR
BEGIN

REGION Network 1: Convert Date to String
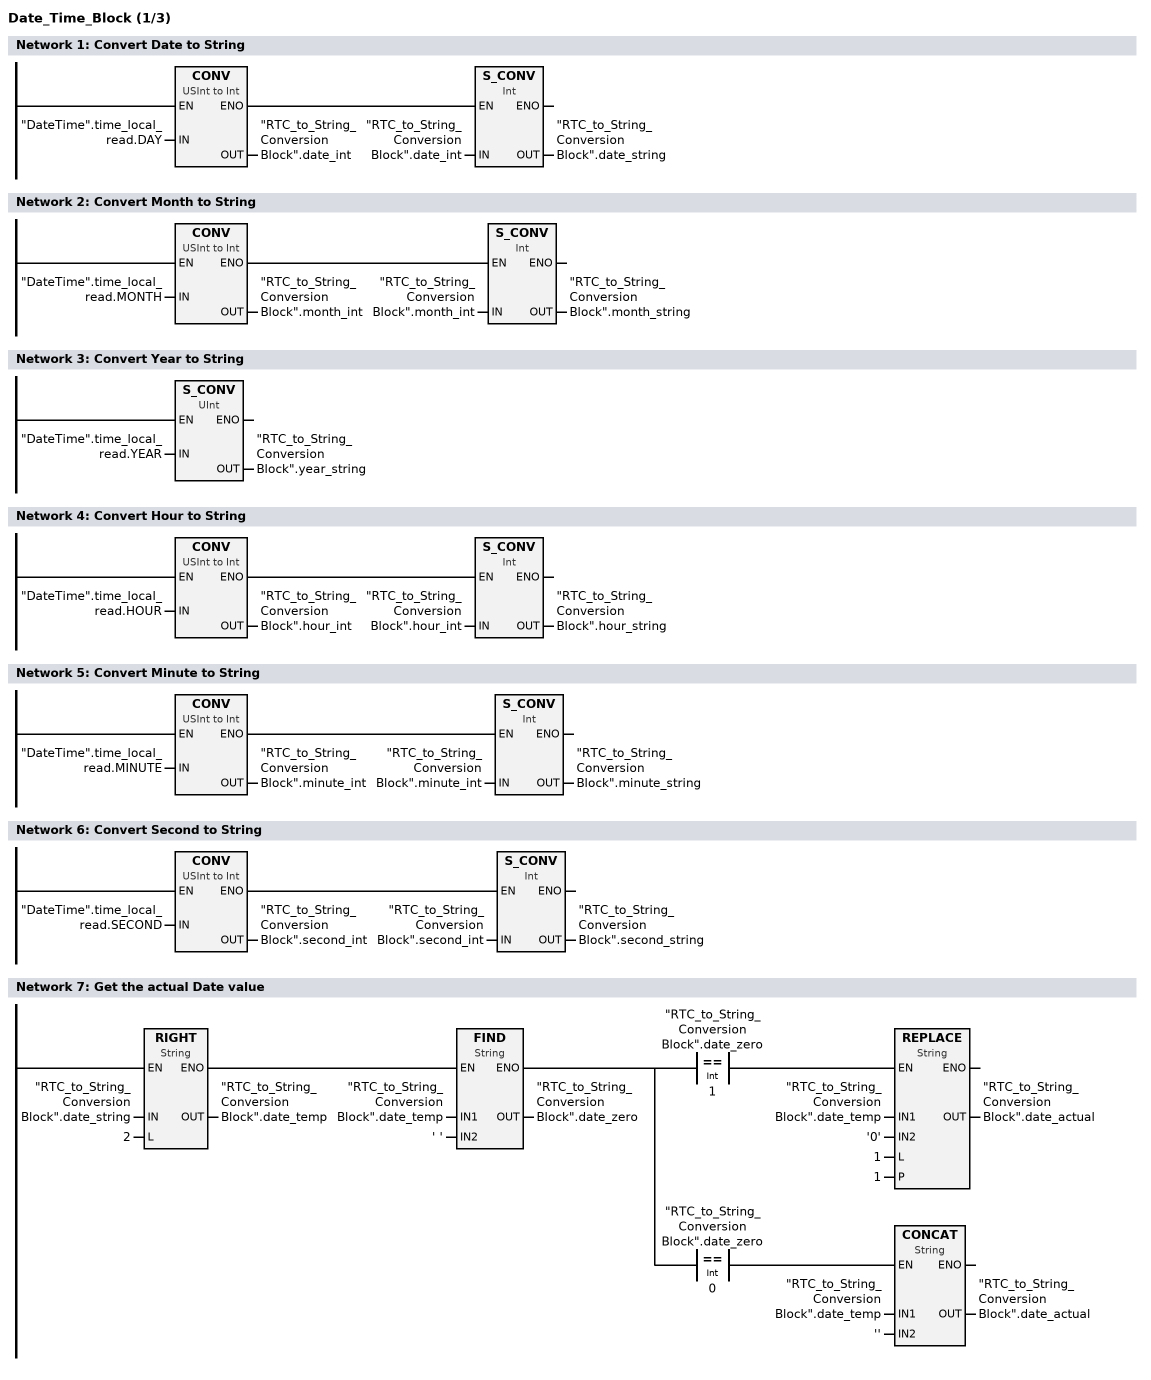
   RUNG wire#powerrail
      { S7_Templates := "[SrcType := USInt, DestType := Int]"; S7_GenerateENO := "TRUE" } Convert(in := "DateTime".time_local_read.DAY, out => "RTC_to_String_Conversion Block".date_int)
      { S7_Templates := "[src_type := Int, dest_type := String]" } S_CONV(IN := "RTC_to_String_Conversion Block".date_int, OUT => "RTC_to_String_Conversion Block".date_string)
   END_RUNG
   // the same network as SCL:
   // ENO of a box is taken as its EN; it also drops when the box reports an error
   "RTC_to_String_Conversion Block".date_int := USINT_TO_INT("DateTime".time_local_read.DAY);
   S_CONV(IN := "RTC_to_String_Conversion Block".date_int, OUT => "RTC_to_String_Conversion Block".date_string);
END_REGION

REGION Network 2: Convert Month to String
   RUNG wire#powerrail
      { S7_Templates := "[SrcType := USInt, DestType := Int]"; S7_GenerateENO := "TRUE" } Convert(in := "DateTime".time_local_read.MONTH, out => "RTC_to_String_Conversion Block".month_int)
      { S7_Templates := "[src_type := Int, dest_type := String]" } S_CONV(IN := "RTC_to_String_Conversion Block".month_int, OUT => "RTC_to_String_Conversion Block".month_string)
   END_RUNG
   // the same network as SCL:
   // ENO of a box is taken as its EN; it also drops when the box reports an error
   "RTC_to_String_Conversion Block".month_int := USINT_TO_INT("DateTime".time_local_read.MONTH);
   S_CONV(IN := "RTC_to_String_Conversion Block".month_int,
          OUT => "RTC_to_String_Conversion Block".month_string);
END_REGION

REGION Network 3: Convert Year to String
   RUNG wire#powerrail
      { S7_Templates := "[src_type := UInt, dest_type := String]" } S_CONV(IN := "DateTime".time_local_read.YEAR, OUT => "RTC_to_String_Conversion Block".year_string)
   END_RUNG
   // the same network as SCL:
   S_CONV(IN := "DateTime".time_local_read.YEAR, OUT => "RTC_to_String_Conversion Block".year_string);
END_REGION

REGION Network 4: Convert Hour to String
   RUNG wire#powerrail
      { S7_Templates := "[SrcType := USInt, DestType := Int]"; S7_GenerateENO := "TRUE" } Convert(in := "DateTime".time_local_read.HOUR, out => "RTC_to_String_Conversion Block".hour_int)
      { S7_Templates := "[src_type := Int, dest_type := String]" } S_CONV(IN := "RTC_to_String_Conversion Block".hour_int, OUT => "RTC_to_String_Conversion Block".hour_string)
   END_RUNG
   // the same network as SCL:
   // ENO of a box is taken as its EN; it also drops when the box reports an error
   "RTC_to_String_Conversion Block".hour_int := USINT_TO_INT("DateTime".time_local_read.HOUR);
   S_CONV(IN := "RTC_to_String_Conversion Block".hour_int, OUT => "RTC_to_String_Conversion Block".hour_string);
END_REGION

REGION Network 5: Convert Minute to String
   RUNG wire#powerrail
      { S7_Templates := "[SrcType := USInt, DestType := Int]"; S7_GenerateENO := "TRUE" } Convert(in := "DateTime".time_local_read.MINUTE, out => "RTC_to_String_Conversion Block".minute_int)
      { S7_Templates := "[src_type := Int, dest_type := String]" } S_CONV(IN := "RTC_to_String_Conversion Block".minute_int, OUT => "RTC_to_String_Conversion Block".minute_string)
   END_RUNG
   // the same network as SCL:
   // ENO of a box is taken as its EN; it also drops when the box reports an error
   "RTC_to_String_Conversion Block".minute_int := USINT_TO_INT("DateTime".time_local_read.MINUTE);
   S_CONV(IN := "RTC_to_String_Conversion Block".minute_int,
          OUT => "RTC_to_String_Conversion Block".minute_string);
END_REGION

REGION Network 6: Convert Second to String
   RUNG wire#powerrail
      { S7_Templates := "[SrcType := USInt, DestType := Int]"; S7_GenerateENO := "TRUE" } Convert(in := "DateTime".time_local_read.SECOND, out => "RTC_to_String_Conversion Block".second_int)
      { S7_Templates := "[src_type := Int, dest_type := String]" } S_CONV(IN := "RTC_to_String_Conversion Block".second_int, OUT => "RTC_to_String_Conversion Block".second_string)
   END_RUNG
   // the same network as SCL:
   // ENO of a box is taken as its EN; it also drops when the box reports an error
   "RTC_to_String_Conversion Block".second_int := USINT_TO_INT("DateTime".time_local_read.SECOND);
   S_CONV(IN := "RTC_to_String_Conversion Block".second_int,
          OUT => "RTC_to_String_Conversion Block".second_string);
END_REGION

REGION Network 7: Get the actual Date value
   RUNG wire#powerrail
      { S7_Templates := "str_type := String" } RIGHT(IN := "RTC_to_String_Conversion Block".date_string, L := 2, OUT => "RTC_to_String_Conversion Block".date_temp)
      { S7_Templates := "str_type := String" } FIND(IN1 := "RTC_to_String_Conversion Block".date_temp, IN2 := ' ', OUT => "RTC_to_String_Conversion Block".date_zero)
      wire#w1
      { S7_Templates := "SrcType := Int" } EQ_Contact(in1 := "RTC_to_String_Conversion Block".date_zero, in2 := 1)
      { S7_Templates := "str_type := String" } REPLACE(IN1 := "RTC_to_String_Conversion Block".date_temp, IN2 := '0', L := 1, P := 1, OUT => "RTC_to_String_Conversion Block".date_actual)
   END_RUNG
   RUNG wire#w1
      { S7_Templates := "SrcType := Int" } EQ_Contact(in1 := "RTC_to_String_Conversion Block".date_zero, in2 := 0)
      { S7_Templates := "[card := 2, str_type := String]" } CONCAT(IN1 := "RTC_to_String_Conversion Block".date_temp, IN2 := '', OUT => "RTC_to_String_Conversion Block".date_actual)
   END_RUNG
   // the same network as SCL:
   RIGHT(IN := "RTC_to_String_Conversion Block".date_string,
         L := 2,
         OUT => "RTC_to_String_Conversion Block".date_temp,
         ENO => #_w1);
   FIND(EN := #_w1,
        IN1 := "RTC_to_String_Conversion Block".date_temp,
        IN2 := ' ',
        OUT => "RTC_to_String_Conversion Block".date_zero,
        ENO => #_w2);
   IF #_w2 AND ("RTC_to_String_Conversion Block".date_zero = 1) THEN
       REPLACE(IN1 := "RTC_to_String_Conversion Block".date_temp,
               IN2 := '0',
               L := 1,
               P := 1,
               OUT => "RTC_to_String_Conversion Block".date_actual);
   END_IF;
   IF #_w2 AND ("RTC_to_String_Conversion Block".date_zero = 0) THEN
       CONCAT(IN1 := "RTC_to_String_Conversion Block".date_temp,
              IN2 := '',
              OUT => "RTC_to_String_Conversion Block".date_actual);
   END_IF;
END_REGION

REGION Network 8: Get the actual month value
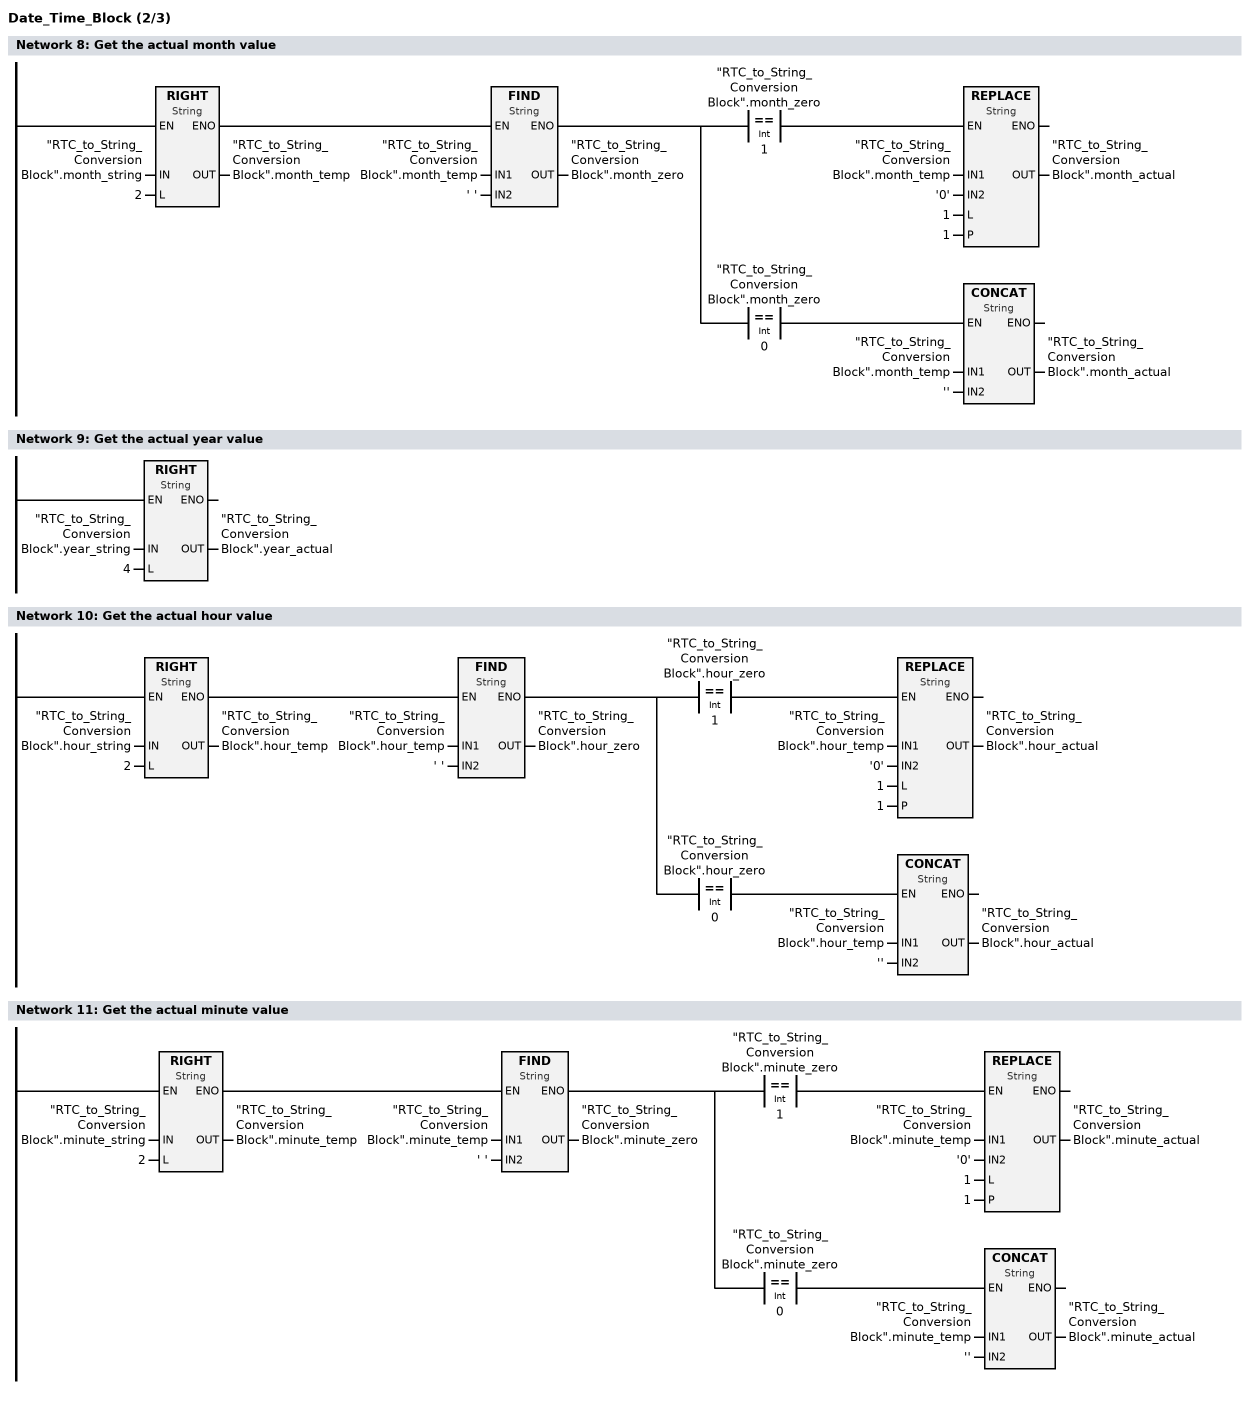
   RUNG wire#powerrail
      { S7_Templates := "str_type := String" } RIGHT(IN := "RTC_to_String_Conversion Block".month_string, L := 2, OUT => "RTC_to_String_Conversion Block".month_temp)
      { S7_Templates := "str_type := String" } FIND(IN1 := "RTC_to_String_Conversion Block".month_temp, IN2 := ' ', OUT => "RTC_to_String_Conversion Block".month_zero)
      wire#w1
      { S7_Templates := "SrcType := Int" } EQ_Contact(in1 := "RTC_to_String_Conversion Block".month_zero, in2 := 1)
      { S7_Templates := "str_type := String" } REPLACE(IN1 := "RTC_to_String_Conversion Block".month_temp, IN2 := '0', L := 1, P := 1, OUT => "RTC_to_String_Conversion Block".month_actual)
   END_RUNG
   RUNG wire#w1
      { S7_Templates := "SrcType := Int" } EQ_Contact(in1 := "RTC_to_String_Conversion Block".month_zero, in2 := 0)
      { S7_Templates := "[card := 2, str_type := String]" } CONCAT(IN1 := "RTC_to_String_Conversion Block".month_temp, IN2 := '', OUT => "RTC_to_String_Conversion Block".month_actual)
   END_RUNG
   // the same network as SCL:
   RIGHT(IN := "RTC_to_String_Conversion Block".month_string,
         L := 2,
         OUT => "RTC_to_String_Conversion Block".month_temp,
         ENO => #_w1);
   FIND(EN := #_w1,
        IN1 := "RTC_to_String_Conversion Block".month_temp,
        IN2 := ' ',
        OUT => "RTC_to_String_Conversion Block".month_zero,
        ENO => #_w2);
   IF #_w2 AND ("RTC_to_String_Conversion Block".month_zero = 1) THEN
       REPLACE(IN1 := "RTC_to_String_Conversion Block".month_temp,
               IN2 := '0',
               L := 1,
               P := 1,
               OUT => "RTC_to_String_Conversion Block".month_actual);
   END_IF;
   IF #_w2 AND ("RTC_to_String_Conversion Block".month_zero = 0) THEN
       CONCAT(IN1 := "RTC_to_String_Conversion Block".month_temp,
              IN2 := '',
              OUT => "RTC_to_String_Conversion Block".month_actual);
   END_IF;
END_REGION

REGION Network 9: Get the actual year value
   RUNG wire#powerrail
      { S7_Templates := "str_type := String" } RIGHT(IN := "RTC_to_String_Conversion Block".year_string, L := 4, OUT => "RTC_to_String_Conversion Block".year_actual)
   END_RUNG
   // the same network as SCL:
   RIGHT(IN := "RTC_to_String_Conversion Block".year_string,
         L := 4,
         OUT => "RTC_to_String_Conversion Block".year_actual);
END_REGION

REGION Network 10: Get the actual hour value
   RUNG wire#powerrail
      { S7_Templates := "str_type := String" } RIGHT(IN := "RTC_to_String_Conversion Block".hour_string, L := 2, OUT => "RTC_to_String_Conversion Block".hour_temp)
      { S7_Templates := "str_type := String" } FIND(IN1 := "RTC_to_String_Conversion Block".hour_temp, IN2 := ' ', OUT => "RTC_to_String_Conversion Block".hour_zero)
      wire#w1
      { S7_Templates := "SrcType := Int" } EQ_Contact(in1 := "RTC_to_String_Conversion Block".hour_zero, in2 := 1)
      { S7_Templates := "str_type := String" } REPLACE(IN1 := "RTC_to_String_Conversion Block".hour_temp, IN2 := '0', L := 1, P := 1, OUT => "RTC_to_String_Conversion Block".hour_actual)
   END_RUNG
   RUNG wire#w1
      { S7_Templates := "SrcType := Int" } EQ_Contact(in1 := "RTC_to_String_Conversion Block".hour_zero, in2 := 0)
      { S7_Templates := "[card := 2, str_type := String]" } CONCAT(IN1 := "RTC_to_String_Conversion Block".hour_temp, IN2 := '', OUT => "RTC_to_String_Conversion Block".hour_actual)
   END_RUNG
   // the same network as SCL:
   RIGHT(IN := "RTC_to_String_Conversion Block".hour_string,
         L := 2,
         OUT => "RTC_to_String_Conversion Block".hour_temp,
         ENO => #_w1);
   FIND(EN := #_w1,
        IN1 := "RTC_to_String_Conversion Block".hour_temp,
        IN2 := ' ',
        OUT => "RTC_to_String_Conversion Block".hour_zero,
        ENO => #_w2);
   IF #_w2 AND ("RTC_to_String_Conversion Block".hour_zero = 1) THEN
       REPLACE(IN1 := "RTC_to_String_Conversion Block".hour_temp,
               IN2 := '0',
               L := 1,
               P := 1,
               OUT => "RTC_to_String_Conversion Block".hour_actual);
   END_IF;
   IF #_w2 AND ("RTC_to_String_Conversion Block".hour_zero = 0) THEN
       CONCAT(IN1 := "RTC_to_String_Conversion Block".hour_temp,
              IN2 := '',
              OUT => "RTC_to_String_Conversion Block".hour_actual);
   END_IF;
END_REGION

REGION Network 11: Get the actual minute value
   RUNG wire#powerrail
      { S7_Templates := "str_type := String" } RIGHT(IN := "RTC_to_String_Conversion Block".minute_string, L := 2, OUT => "RTC_to_String_Conversion Block".minute_temp)
      { S7_Templates := "str_type := String" } FIND(IN1 := "RTC_to_String_Conversion Block".minute_temp, IN2 := ' ', OUT => "RTC_to_String_Conversion Block".minute_zero)
      wire#w1
      { S7_Templates := "SrcType := Int" } EQ_Contact(in1 := "RTC_to_String_Conversion Block".minute_zero, in2 := 1)
      { S7_Templates := "str_type := String" } REPLACE(IN1 := "RTC_to_String_Conversion Block".minute_temp, IN2 := '0', L := 1, P := 1, OUT => "RTC_to_String_Conversion Block".minute_actual)
   END_RUNG
   RUNG wire#w1
      { S7_Templates := "SrcType := Int" } EQ_Contact(in1 := "RTC_to_String_Conversion Block".minute_zero, in2 := 0)
      { S7_Templates := "[card := 2, str_type := String]" } CONCAT(IN1 := "RTC_to_String_Conversion Block".minute_temp, IN2 := '', OUT => "RTC_to_String_Conversion Block".minute_actual)
   END_RUNG
   // the same network as SCL:
   RIGHT(IN := "RTC_to_String_Conversion Block".minute_string,
         L := 2,
         OUT => "RTC_to_String_Conversion Block".minute_temp,
         ENO => #_w1);
   FIND(EN := #_w1,
        IN1 := "RTC_to_String_Conversion Block".minute_temp,
        IN2 := ' ',
        OUT => "RTC_to_String_Conversion Block".minute_zero,
        ENO => #_w2);
   IF #_w2 AND ("RTC_to_String_Conversion Block".minute_zero = 1) THEN
       REPLACE(IN1 := "RTC_to_String_Conversion Block".minute_temp,
               IN2 := '0',
               L := 1,
               P := 1,
               OUT => "RTC_to_String_Conversion Block".minute_actual);
   END_IF;
   IF #_w2 AND ("RTC_to_String_Conversion Block".minute_zero = 0) THEN
       CONCAT(IN1 := "RTC_to_String_Conversion Block".minute_temp,
              IN2 := '',
              OUT => "RTC_to_String_Conversion Block".minute_actual);
   END_IF;
END_REGION

REGION Network 12: Get the actual second value
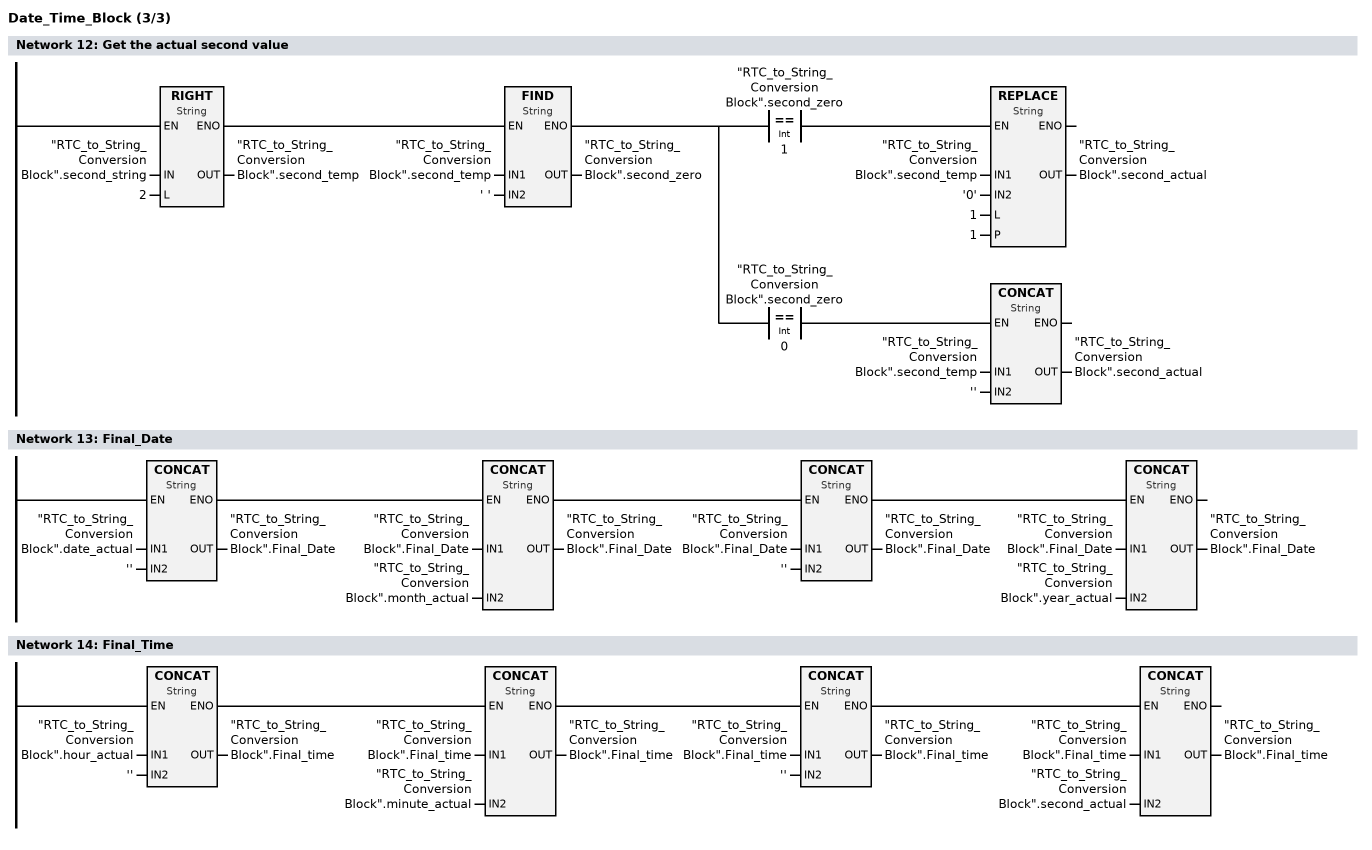
   RUNG wire#powerrail
      { S7_Templates := "str_type := String" } RIGHT(IN := "RTC_to_String_Conversion Block".second_string, L := 2, OUT => "RTC_to_String_Conversion Block".second_temp)
      { S7_Templates := "str_type := String" } FIND(IN1 := "RTC_to_String_Conversion Block".second_temp, IN2 := ' ', OUT => "RTC_to_String_Conversion Block".second_zero)
      wire#w1
      { S7_Templates := "SrcType := Int" } EQ_Contact(in1 := "RTC_to_String_Conversion Block".second_zero, in2 := 1)
      { S7_Templates := "str_type := String" } REPLACE(IN1 := "RTC_to_String_Conversion Block".second_temp, IN2 := '0', L := 1, P := 1, OUT => "RTC_to_String_Conversion Block".second_actual)
   END_RUNG
   RUNG wire#w1
      { S7_Templates := "SrcType := Int" } EQ_Contact(in1 := "RTC_to_String_Conversion Block".second_zero, in2 := 0)
      { S7_Templates := "[card := 2, str_type := String]" } CONCAT(IN1 := "RTC_to_String_Conversion Block".second_temp, IN2 := '', OUT => "RTC_to_String_Conversion Block".second_actual)
   END_RUNG
   // the same network as SCL:
   RIGHT(IN := "RTC_to_String_Conversion Block".second_string,
         L := 2,
         OUT => "RTC_to_String_Conversion Block".second_temp,
         ENO => #_w1);
   FIND(EN := #_w1,
        IN1 := "RTC_to_String_Conversion Block".second_temp,
        IN2 := ' ',
        OUT => "RTC_to_String_Conversion Block".second_zero,
        ENO => #_w2);
   IF #_w2 AND ("RTC_to_String_Conversion Block".second_zero = 1) THEN
       REPLACE(IN1 := "RTC_to_String_Conversion Block".second_temp,
               IN2 := '0',
               L := 1,
               P := 1,
               OUT => "RTC_to_String_Conversion Block".second_actual);
   END_IF;
   IF #_w2 AND ("RTC_to_String_Conversion Block".second_zero = 0) THEN
       CONCAT(IN1 := "RTC_to_String_Conversion Block".second_temp,
              IN2 := '',
              OUT => "RTC_to_String_Conversion Block".second_actual);
   END_IF;
END_REGION

REGION Network 13: Final_Date
   RUNG wire#powerrail
      { S7_Templates := "[card := 2, str_type := String]" } CONCAT(IN1 := "RTC_to_String_Conversion Block".date_actual, IN2 := '', OUT => "RTC_to_String_Conversion Block".Final_Date)
      { S7_Templates := "[card := 2, str_type := String]" } CONCAT(IN1 := "RTC_to_String_Conversion Block".Final_Date, IN2 := "RTC_to_String_Conversion Block".month_actual, OUT => "RTC_to_String_Conversion Block".Final_Date)
      { S7_Templates := "[card := 2, str_type := String]" } CONCAT(IN1 := "RTC_to_String_Conversion Block".Final_Date, IN2 := '', OUT => "RTC_to_String_Conversion Block".Final_Date)
      { S7_Templates := "[card := 2, str_type := String]" } CONCAT(IN1 := "RTC_to_String_Conversion Block".Final_Date, IN2 := "RTC_to_String_Conversion Block".year_actual, OUT => "RTC_to_String_Conversion Block".Final_Date)
   END_RUNG
   // the same network as SCL:
   CONCAT(IN1 := "RTC_to_String_Conversion Block".date_actual,
          IN2 := '',
          OUT => "RTC_to_String_Conversion Block".Final_Date,
          ENO => #_w1);
   CONCAT(EN := #_w1,
          IN1 := "RTC_to_String_Conversion Block".Final_Date,
          IN2 := "RTC_to_String_Conversion Block".month_actual,
          OUT => "RTC_to_String_Conversion Block".Final_Date,
          ENO => #_w2);
   CONCAT(EN := #_w2,
          IN1 := "RTC_to_String_Conversion Block".Final_Date,
          IN2 := '',
          OUT => "RTC_to_String_Conversion Block".Final_Date,
          ENO => #_w3);
   IF #_w3 THEN
       CONCAT(IN1 := "RTC_to_String_Conversion Block".Final_Date,
              IN2 := "RTC_to_String_Conversion Block".year_actual,
              OUT => "RTC_to_String_Conversion Block".Final_Date);
   END_IF;
END_REGION

REGION Network 14: Final_Time
   RUNG wire#powerrail
      { S7_Templates := "[card := 2, str_type := String]" } CONCAT(IN1 := "RTC_to_String_Conversion Block".hour_actual, IN2 := '', OUT => "RTC_to_String_Conversion Block".Final_time)
      { S7_Templates := "[card := 2, str_type := String]" } CONCAT(IN1 := "RTC_to_String_Conversion Block".Final_time, IN2 := "RTC_to_String_Conversion Block".minute_actual, OUT => "RTC_to_String_Conversion Block".Final_time)
      { S7_Templates := "[card := 2, str_type := String]" } CONCAT(IN1 := "RTC_to_String_Conversion Block".Final_time, IN2 := '', OUT => "RTC_to_String_Conversion Block".Final_time)
      { S7_Templates := "[card := 2, str_type := String]" } CONCAT(IN1 := "RTC_to_String_Conversion Block".Final_time, IN2 := "RTC_to_String_Conversion Block".second_actual, OUT => "RTC_to_String_Conversion Block".Final_time)
   END_RUNG
   // the same network as SCL:
   CONCAT(IN1 := "RTC_to_String_Conversion Block".hour_actual,
          IN2 := '',
          OUT => "RTC_to_String_Conversion Block".Final_time,
          ENO => #_w1);
   CONCAT(EN := #_w1,
          IN1 := "RTC_to_String_Conversion Block".Final_time,
          IN2 := "RTC_to_String_Conversion Block".minute_actual,
          OUT => "RTC_to_String_Conversion Block".Final_time,
          ENO => #_w2);
   CONCAT(EN := #_w2,
          IN1 := "RTC_to_String_Conversion Block".Final_time,
          IN2 := '',
          OUT => "RTC_to_String_Conversion Block".Final_time,
          ENO => #_w3);
   IF #_w3 THEN
       CONCAT(IN1 := "RTC_to_String_Conversion Block".Final_time,
              IN2 := "RTC_to_String_Conversion Block".second_actual,
              OUT => "RTC_to_String_Conversion Block".Final_time);
   END_IF;
END_REGION
END_ORGANIZATION_BLOCK

ORGANIZATION_BLOCK "PidCyclicInterrupt"   // OB30, LAD, CyclicInterrupt
{ S7_Optimized_Access := 'TRUE' }
// stored: CyclicTime 50000, SetENOAutomatically false
BEGIN

REGION Network 1: "Fv1-Cv01" PID Block
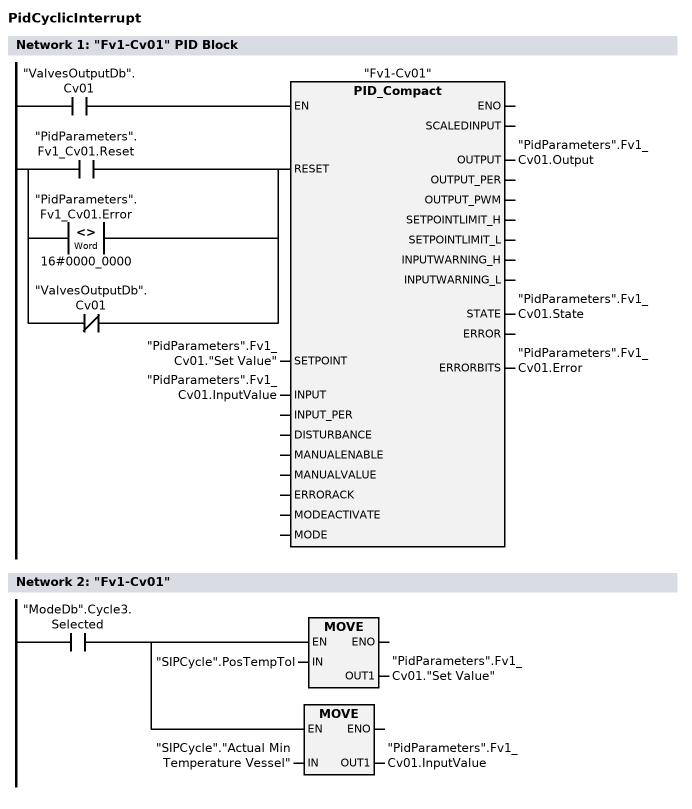
   RUNG wire#powerrail
      Contact( "ValvesOutputDb".Cv01 )
      "Fv1-Cv01".PID_Compact(Reset := wire#w1, Setpoint := "PidParameters".Fv1_Cv01."Set Value", Input := "PidParameters".Fv1_Cv01.InputValue, Input_PER :=, Disturbance :=, ManualEnable :=, ManualValue :=, ErrorAck :=, ModeActivate :=, Mode :=, ScaledInput =>, Output => "PidParameters".Fv1_Cv01.Output, Output_PER =>, Output_PWM =>, SetpointLimit_H =>, SetpointLimit_L =>, InputWarning_H =>, InputWarning_L =>, State => "PidParameters".Fv1_Cv01.State, Error =>, ErrorBits => "PidParameters".Fv1_Cv01.Error)
   END_RUNG
   RUNG wire#powerrail
      Contact( "PidParameters".Fv1_Cv01.Reset )
   END_RUNG wire#w1
   RUNG wire#powerrail
      { S7_Templates := "SrcType := Word" } NE_Contact(in1 := "PidParameters".Fv1_Cv01.Error, in2 := 16#0000_0000)
   END_RUNG wire#w1
   RUNG wire#powerrail
      I_Contact( "ValvesOutputDb".Cv01 )
   END_RUNG wire#w1
   // the same network as SCL:
   IF "ValvesOutputDb".Cv01 THEN
       "Fv1-Cv01"(Reset := "PidParameters".Fv1_Cv01.Reset OR ("PidParameters".Fv1_Cv01.Error <> 16#0000_0000) OR NOT "ValvesOutputDb".Cv01,   // PID_Compact
                  Setpoint := "PidParameters".Fv1_Cv01."Set Value",
                  Input := "PidParameters".Fv1_Cv01.InputValue,
                  Output => "PidParameters".Fv1_Cv01.Output,
                  State => "PidParameters".Fv1_Cv01.State,
                  ErrorBits => "PidParameters".Fv1_Cv01.Error);
   END_IF;
END_REGION

REGION Network 2: "Fv1-Cv01"
   RUNG wire#powerrail
      Contact( "ModeDb".Cycle3.Selected )
      wire#w1
      Move(in := "SIPCycle".PosTempTol, out1 => "PidParameters".Fv1_Cv01."Set Value")
   END_RUNG
   RUNG wire#w1
      Move(in := "SIPCycle"."Actual Min Temperature Vessel", out1 => "PidParameters".Fv1_Cv01.InputValue)
   END_RUNG
   // the same network as SCL:
   IF "ModeDb".Cycle3.Selected THEN
       "PidParameters".Fv1_Cv01."Set Value" := "SIPCycle".PosTempTol;
       "PidParameters".Fv1_Cv01.InputValue := "SIPCycle"."Actual Min Temperature Vessel";
   END_IF;
END_REGION
END_ORGANIZATION_BLOCK

FUNCTION_BLOCK "BatchDetailsLength"   // FB99, LAD
{ S7_Optimized_Access := 'TRUE' }
// stored: AutoNumber false, MemoryReserve 100, SetENOAutomatically false
   VAR_OUTPUT
      EquipmentID_Len { ExternalAccessible := 'False'; ExternalVisible := 'False'; ExternalWritable := 'False'} : Int;
      ProductName_Len { ExternalAccessible := 'False'; ExternalVisible := 'False'; ExternalWritable := 'False'} : Int;
      BatchNum_Len { ExternalAccessible := 'False'; ExternalVisible := 'False'; ExternalWritable := 'False'} : Int;
      PrintInt_Len { ExternalAccessible := 'False'; ExternalVisible := 'False'; ExternalWritable := 'False'} : Int;
   END_VAR
   VAR_TEMP   // added for the SCL form of the ladder/FBD networks
      _w1 : Bool;
      _w2 : Bool;
   END_VAR
BEGIN

REGION Network 1: BATCH DETAIL LENGTH
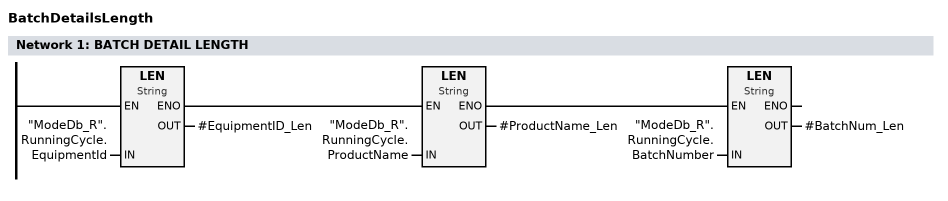
   RUNG wire#powerrail
      { S7_Templates := "[str_type := String, return_type := Int]" } LEN(IN := "ModeDb_R".RunningCycle.EquipmentId, OUT => #EquipmentID_Len)
      { S7_Templates := "[str_type := String, return_type := Int]" } LEN(IN := "ModeDb_R".RunningCycle.ProductName, OUT => #ProductName_Len)
      { S7_Templates := "[str_type := String, return_type := Int]" } LEN(IN := "ModeDb_R".RunningCycle.BatchNumber, OUT => #BatchNum_Len)
   END_RUNG
   // the same network as SCL:
   LEN(IN := "ModeDb_R".RunningCycle.EquipmentId, OUT => #EquipmentID_Len, ENO => #_w1);
   LEN(EN := #_w1, IN := "ModeDb_R".RunningCycle.ProductName, OUT => #ProductName_Len, ENO => #_w2);
   IF #_w2 THEN LEN(IN := "ModeDb_R".RunningCycle.BatchNumber, OUT => #BatchNum_Len); END_IF;
END_REGION
END_FUNCTION_BLOCK

FUNCTION_BLOCK "FB1"   // FB8, LAD
{ S7_Optimized_Access := 'FALSE' }
// stored: AutoNumber false, SetENOAutomatically false
   VAR_INPUT
      TIME_START : Bool;
      TIME_PULSE : Bool;
      TIME_TRSET : Bool;
      MINI_ENABLE : Bool;
      TIME_IN_MINI : Int;
      TIME_IN_SEC : Int;
   END_VAR
   VAR_OUTPUT
      DONE_BIT : Bool;
      ES_MINIT : DInt;
      ES_SEC : DInt;
   END_VAR
   VAR_IN_OUT
      TEMP_1 : Int;
      TEMP_5 : Int;
      TEMP_2 : Int;
      TEMP_3 : Int;
      TEMP_4 : DInt;
      TEMP_BIT_1 : Bool;
   END_VAR
BEGIN

REGION Network 1
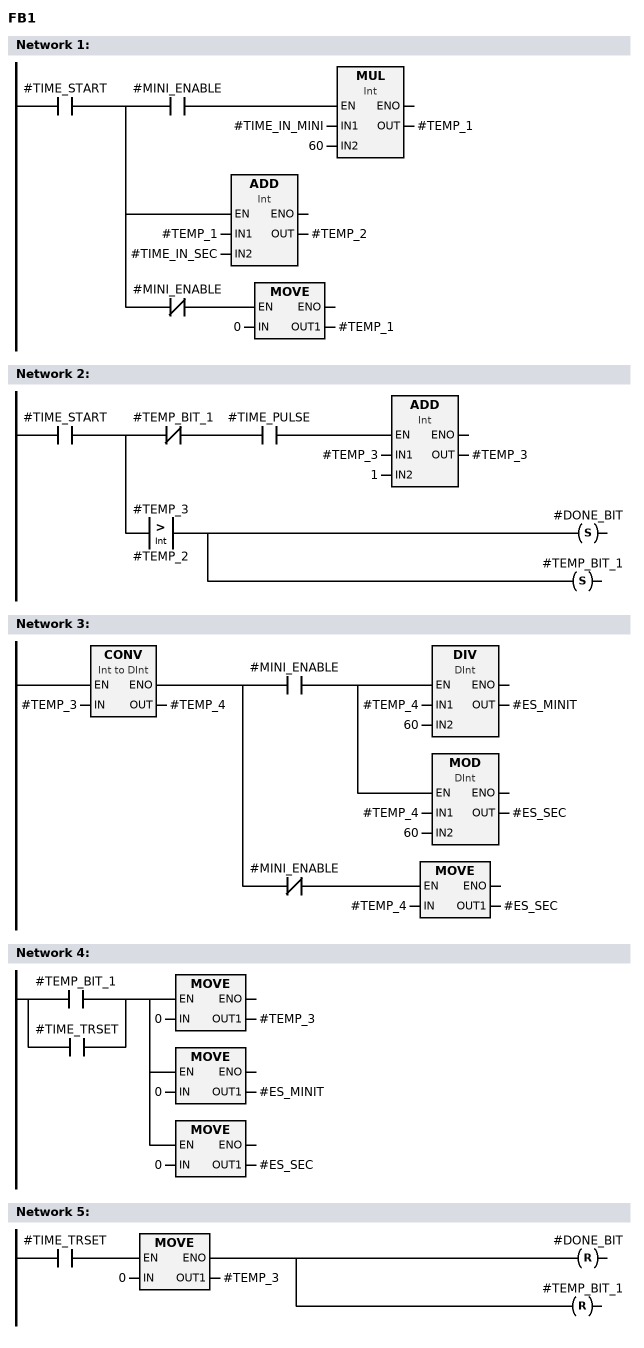
   RUNG wire#powerrail
      Contact( #TIME_START )
      wire#w1
      Contact( #MINI_ENABLE )
      { S7_Templates := "SrcType := Int"; S7_GenerateENO := "TRUE" } Mul(in1 := #TIME_IN_MINI, in2 := 60, out => #TEMP_1)
   END_RUNG
   RUNG wire#w1
      { S7_Templates := "SrcType := Int"; S7_GenerateENO := "TRUE" } Add(in1 := #TEMP_1, in2 := #TIME_IN_SEC, out => #TEMP_2)
   END_RUNG
   RUNG wire#w1
      I_Contact( #MINI_ENABLE )
      { S7_GenerateENO := "TRUE" } Move(in := 0, out1 => #TEMP_1)
   END_RUNG
   // the same network as SCL:
   IF #TIME_START AND #MINI_ENABLE THEN #TEMP_1 := #TIME_IN_MINI * 60; END_IF;
   IF #TIME_START THEN #TEMP_2 := #TEMP_1 + #TIME_IN_SEC; END_IF;
   IF #TIME_START AND NOT #MINI_ENABLE THEN #TEMP_1 := 0; END_IF;
END_REGION

REGION Network 2
   RUNG wire#powerrail
      Contact( #TIME_START )
      wire#w1
      I_Contact( #TEMP_BIT_1 )
      Contact( #TIME_PULSE )
      { S7_Templates := "SrcType := Int"; S7_GenerateENO := "TRUE" } Add(in1 := #TEMP_3, in2 := 1, out => #TEMP_3)
   END_RUNG
   RUNG wire#w1
      { S7_Templates := "SrcType := Int" } GT_Contact(in1 := #TEMP_3, in2 := #TEMP_2)
      wire#w2
      S_Coil( #DONE_BIT )
   END_RUNG
   RUNG wire#w2
      S_Coil( #TEMP_BIT_1 )
   END_RUNG
   // the same network as SCL:
   IF #TIME_START AND NOT #TEMP_BIT_1 AND #TIME_PULSE THEN #TEMP_3 := #TEMP_3 + 1; END_IF;
   IF #TIME_START AND (#TEMP_3 > #TEMP_2) THEN
       #DONE_BIT := TRUE;
       #TEMP_BIT_1 := TRUE;
   END_IF;
END_REGION

REGION Network 3
   RUNG wire#powerrail
      { S7_Templates := "[SrcType := Int, DestType := DInt]"; S7_GenerateENO := "TRUE" } Convert(in := #TEMP_3, out => #TEMP_4)
      wire#w1
      Contact( #MINI_ENABLE )
      wire#w2
      { S7_Templates := "SrcType := DInt"; S7_GenerateENO := "TRUE" } Div(in1 := #TEMP_4, in2 := 60, out => #ES_MINIT)
   END_RUNG
   RUNG wire#w2
      { S7_Templates := "SrcType := DInt"; S7_GenerateENO := "TRUE" } Mod(in1 := #TEMP_4, in2 := 60, out => #ES_SEC)
   END_RUNG
   RUNG wire#w1
      I_Contact( #MINI_ENABLE )
      { S7_GenerateENO := "TRUE" } Move(in := #TEMP_4, out1 => #ES_SEC)
   END_RUNG
   // the same network as SCL:
   // ENO of a box is taken as its EN; it also drops when the box reports an error
   #TEMP_4 := INT_TO_DINT(#TEMP_3);
   IF #MINI_ENABLE THEN
       #ES_MINIT := #TEMP_4 / 60;
       #ES_SEC := #TEMP_4 MOD 60;
   END_IF;
   IF NOT #MINI_ENABLE THEN #ES_SEC := #TEMP_4; END_IF;
END_REGION

REGION Network 4
   RUNG wire#powerrail
      Contact( #TEMP_BIT_1 )
      wire#w1
      { S7_GenerateENO := "TRUE" } Move(in := 0, out1 => #TEMP_3)
   END_RUNG
   RUNG wire#powerrail
      Contact( #TIME_TRSET )
   END_RUNG wire#w1
   RUNG wire#w1
      { S7_GenerateENO := "TRUE" } Move(in := 0, out1 => #ES_MINIT)
   END_RUNG
   RUNG wire#w1
      { S7_GenerateENO := "TRUE" } Move(in := 0, out1 => #ES_SEC)
   END_RUNG
   // the same network as SCL:
   IF #TEMP_BIT_1 OR #TIME_TRSET THEN
       #TEMP_3 := 0;
       #ES_MINIT := 0;
       #ES_SEC := 0;
   END_IF;
END_REGION

REGION Network 5
   RUNG wire#powerrail
      Contact( #TIME_TRSET )
      { S7_GenerateENO := "TRUE" } Move(in := 0, out1 => #TEMP_3)
      wire#w1
      R_Coil( #DONE_BIT )
   END_RUNG
   RUNG wire#w1
      R_Coil( #TEMP_BIT_1 )
   END_RUNG
   // the same network as SCL:
   // ENO of a box is taken as its EN; it also drops when the box reports an error
   IF #TIME_TRSET THEN
       #TEMP_3 := 0;
       #DONE_BIT := FALSE;
       #TEMP_BIT_1 := FALSE;
   END_IF;
END_REGION
END_FUNCTION_BLOCK

FUNCTION_BLOCK "Motor Block"   // FB3, LAD
{ S7_Optimized_Access := 'FALSE' }
// stored: AutoNumber false, SetENOAutomatically false
   VAR_INPUT
      Cmd { ExternalVisible := 'False'} : Bool;
      SimulationOn { ExternalVisible := 'False'} : Bool;
      MotorFeedbackInput { ExternalVisible := 'False'} : Bool;
      WaterSensorSelection { ExternalVisible := 'False'} : Bool;
      WaterSensorInput { ExternalVisible := 'False'} : Bool;
      AlwaysTrue : Bool;
      AlwaysFalse : Bool;
      FBCheckDelay { ExternalVisible := 'False'} : Int;
      WSCheckDelay { ExternalVisible := 'False'} : Int;
      secs { ExternalVisible := 'False'} : Bool;
      AlarmAck { ExternalVisible := 'False'} : Bool;
   END_VAR
   VAR_OUTPUT
      Output { ExternalVisible := 'False'} : Bool;
      FeedBackTripAlarm : Bool;
      NoWaterFlowAlarm : Bool;
   END_VAR
   VAR_IN_OUT
      OpFbTrip { ExternalVisible := 'False'} : Bool;
      OpWaterSensorTrip { ExternalVisible := 'False'} : Bool;
      FBCheckActualTime { ExternalVisible := 'False'} : Int;
      WSCheckActualTime { ExternalVisible := 'False'} : Int;
   END_VAR
   VAR_TEMP   // added for the SCL form of the ladder/FBD networks
      _w1 : Bool;
      _w2 : Bool;
   END_VAR
BEGIN

REGION Network 1: OPOn
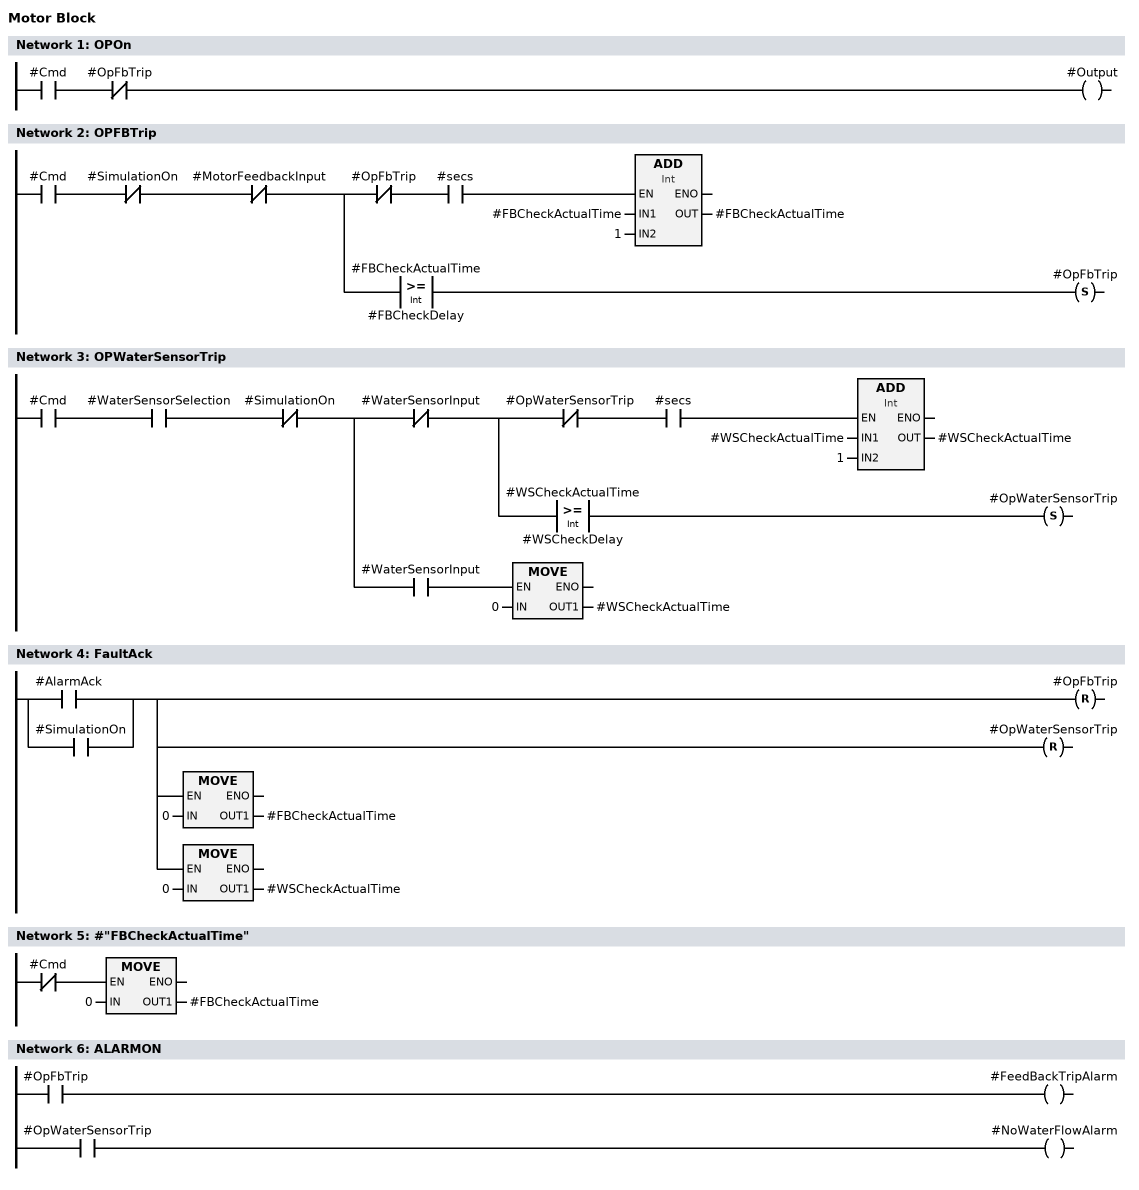
   RUNG wire#powerrail
      Contact( #Cmd )
      I_Contact( #OpFbTrip )
      Coil( #Output )
   END_RUNG
   // the same network as SCL:
   #Output := #Cmd AND NOT #OpFbTrip;
END_REGION

REGION Network 2: OPFBTrip
   RUNG wire#powerrail
      Contact( #Cmd )
      I_Contact( #SimulationOn )
      I_Contact( #MotorFeedbackInput )
      wire#w1
      I_Contact( #OpFbTrip )
      Contact( #secs )
      { S7_Templates := "SrcType := Int"; S7_GenerateENO := "TRUE" } Add(in1 := #FBCheckActualTime, in2 := 1, out => #FBCheckActualTime)
   END_RUNG
   RUNG wire#w1
      { S7_Templates := "SrcType := Int" } GE_Contact(in1 := #FBCheckActualTime, in2 := #FBCheckDelay)
      S_Coil( #OpFbTrip )
   END_RUNG
   // the same network as SCL:
   #_w1 := #Cmd AND NOT #SimulationOn AND NOT #MotorFeedbackInput;
   IF #_w1 AND NOT #OpFbTrip AND #secs THEN #FBCheckActualTime := #FBCheckActualTime + 1; END_IF;
   IF #_w1 AND (#FBCheckActualTime >= #FBCheckDelay) THEN #OpFbTrip := TRUE; END_IF;
END_REGION

REGION Network 3: OPWaterSensorTrip
   RUNG wire#powerrail
      Contact( #Cmd )
      Contact( #WaterSensorSelection )
      I_Contact( #SimulationOn )
      wire#w1
      I_Contact( #WaterSensorInput )
      wire#w2
      I_Contact( #OpWaterSensorTrip )
      Contact( #secs )
      { S7_Templates := "SrcType := Int"; S7_GenerateENO := "TRUE" } Add(in1 := #WSCheckActualTime, in2 := 1, out => #WSCheckActualTime)
   END_RUNG
   RUNG wire#w2
      { S7_Templates := "SrcType := Int" } GE_Contact(in1 := #WSCheckActualTime, in2 := #WSCheckDelay)
      S_Coil( #OpWaterSensorTrip )
   END_RUNG
   RUNG wire#w1
      Contact( #WaterSensorInput )
      { S7_GenerateENO := "TRUE" } Move(in := 0, out1 => #WSCheckActualTime)
   END_RUNG
   // the same network as SCL:
   #_w1 := #Cmd AND #WaterSensorSelection AND NOT #SimulationOn;
   #_w2 := #_w1 AND NOT #WaterSensorInput;
   IF #_w2 AND NOT #OpWaterSensorTrip AND #secs THEN #WSCheckActualTime := #WSCheckActualTime + 1; END_IF;
   IF #_w2 AND (#WSCheckActualTime >= #WSCheckDelay) THEN #OpWaterSensorTrip := TRUE; END_IF;
   IF #_w1 AND #WaterSensorInput THEN #WSCheckActualTime := 0; END_IF;
END_REGION

REGION Network 4: FaultAck
   RUNG wire#powerrail
      Contact( #AlarmAck )
      wire#w1
      R_Coil( #OpFbTrip )
   END_RUNG
   RUNG wire#powerrail
      Contact( #SimulationOn )
   END_RUNG wire#w1
   RUNG wire#w1
      R_Coil( #OpWaterSensorTrip )
   END_RUNG
   RUNG wire#w1
      { S7_GenerateENO := "TRUE" } Move(in := 0, out1 => #FBCheckActualTime)
   END_RUNG
   RUNG wire#w1
      { S7_GenerateENO := "TRUE" } Move(in := 0, out1 => #WSCheckActualTime)
   END_RUNG
   // the same network as SCL:
   IF #AlarmAck OR #SimulationOn THEN
       #OpFbTrip := FALSE;
       #OpWaterSensorTrip := FALSE;
       #FBCheckActualTime := 0;
       #WSCheckActualTime := 0;
   END_IF;
END_REGION

REGION Network 5: #"FBCheckActualTime"
   RUNG wire#powerrail
      I_Contact( #Cmd )
      { S7_GenerateENO := "TRUE" } Move(in := 0, out1 => #FBCheckActualTime)
   END_RUNG
   // the same network as SCL:
   IF NOT #Cmd THEN #FBCheckActualTime := 0; END_IF;
END_REGION

REGION Network 6: ALARMON
   RUNG wire#powerrail
      Contact( #OpFbTrip )
      Coil( #FeedBackTripAlarm )
   END_RUNG
   RUNG wire#powerrail
      Contact( #OpWaterSensorTrip )
      Coil( #NoWaterFlowAlarm )
   END_RUNG
   // the same network as SCL:
   #FeedBackTripAlarm := #OpFbTrip;
   #NoWaterFlowAlarm := #OpWaterSensorTrip;
END_REGION
END_FUNCTION_BLOCK

FUNCTION_BLOCK "SIP Block"   // FB501, LAD
{ S7_Optimized_Access := 'FALSE' }
// stored: AutoNumber false, SetENOAutomatically false
   VAR_INPUT
      secs : Bool;   // secs clock pulse
      "Always On" : Bool;
      "Always Off" : Bool;
      Start : Bool;
      Pause : Bool;
      Abort : Bool;
      "Fault Bit" : Bool;
      "Startup msg Sel" : Bool;   // 0: No; 1 : Yes
      "Startup Ack" : Bool;
      "Pulsing Cycle Active" : Bool;   // 0: No; 1 : Yes
      "Steam purging Active" : Bool;   // 0: No; 1 : Yes
      "Initial pulsing Selection" : Bool;   // 0: Same; 1:Different
      "Sterilization Abort Selection" : Int;   // 0: Restart; 1: Abort; 2: Popup; 3: Repetition
      "Continous/Pressurise Air purge sel" { ExternalAccessible := 'False'; ExternalVisible := 'False'; ExternalWritable := 'False'} : Bool;   // 0: continous ; 1: Pressurise
      "Time/Temperature Air purge sel" : Bool;   // 0: Time ; 1: Temperature
      "Hot air drying sel" : Bool;   // 0: No; 1 : Yes
      "SIP Abort Btn" : Bool;
      "SIP Continue Btn" : Bool;
      "Cooling Msg ACK Btn" : Bool;
      "Final Pressure Selection" : Bool;
      "Steam Purging Time" : Int;
      "No of Pulses" : Int;
      "Pulsing Temperature-1" : Real;
      "Pulsing Temperature-2" : Real;
      "Pulsing Temperature-3" : Real;
      "Pulsing Temperature-4" : Real;
      "Pulsing Temperature-5" : Real;
      "Pulsing Pressure-1" : Real;
      "Pulsing Pressure-2" : Real;
      "Pulsing Pressure-3" : Real;
      "Pulsing Pressure-4" : Real;
      "Pulsing Pressure-5" : Real;
      "Pulsing Low Pressure" : Real;
      "SIP Hold time" : Int;
      "SIP Set temp" : Real;
      "SIP Hold temp" : Real;
      "SIP Reset temp" : Real;
      "SIP High Temp" : Real;
      "SIP Pressure" : Real;
      "Pressure To Start Air Purge" : Real;
      "Hot Drying Time" : Int;
      "Hot Air Set Temperature" : Real;
      "Hot Air Actual Temperature" : Real;
      "Air Cooling High Pressure" : Real;
      "Air Cooling Low Pressure" : Real;
      "Cold Drying End Temperature" : Real;
      "Set Positive Purge Pressure" : Real;
      "Actual Lowest Vessel Pressure" : Real;
      "Actual Highest Vessel Pressure" : Real;
      "Actual Lowest temperature" : Real;
      "Actual Highest Temperature" : Real;
      "Actual vessel Pressure" : Real;
      "Air Purge ack" : Bool;   // Should be high after ack
      "Final Pressure Msg ACK" : Bool;
      "Final JD Required" : Bool := false;   // 0: No; 1 : Yes
      "Safety Pressure" : Real;
      "Cooling Temperature" : Real;
      "JV JD delay" : Int;
      "Sterilization Set Repetition" : Int;
      "Cooling popup Active" : Bool;
      "Alarm Ack" : Bool;
      Printinterval : Int;
   END_VAR
   VAR_OUTPUT
      "Cycle Over" : Bool;
      "Steam Control Valve" : Bool;
      "Hot Air Valves" : Bool;
      "Air Valve" : Bool;
      "Positive Purge Valve" : Bool;
      "Cycle Status" : Int;
      "SIP hold time mins" : DInt;
      "sip hold time secs" : DInt;
      "Abort SIP" : Bool;
      "High Temperature Alarm" : Bool;
      "High Pressure Alarm" : Bool;
      "Low Pressure Alarm" : Bool;
      "Hot Drying Actual Time mins" : DInt;
      "Hot Drying Actual Time secs" : DInt;
      "Start Cooling line" : Bool;
      "Cip drain valves" : Bool;
      "Line Valves-1" : Bool;
      "Line Valves-2" : Bool;
      "Line Valves-3" : Bool;
      "Line Valves-4" : Bool;
      "Drain Valves-1" : Bool;
      "Drain Valves-2" : Bool;
      "Drain Valves-3" : Bool;
      "Drain Valves-4" : Bool;
      "Cycle Status_Str" : String[50];
   END_VAR
   VAR_IN_OUT
      "steam pulsing on" : Bool;
      Running : Bool;
      Selected : Bool;
      "SIP Selected" : Bool;
      "Pulsing Temp Reached" : Bool;
      "Pulsing Temp Reached re" : Bool;
      "SIP Abort or Continue Msg" : Bool;
      "Abort SIP Cycle" : Bool;
      "Reset Hold Timer" : Bool;
      "Cooling Msg" : Bool;
      "Start Jacket Drain After SIP" : Bool;
      "Line Valves" : Bool;
      "Drain Valves" : Bool;
      Abort_Temp : Bool;
      "Actual Pulse" : Int;
      "Start SIP" : Bool;
      "Pulsing Delay Done" : Bool;
      "Start SIP Timer" : Bool;
      "sip done" : Bool;
      "Pause SIP Timer" : Bool;
      temp1 : Bool;
      "Hot Drying Time Over" : Bool;
      "Air Purge Temp Reached" : Bool;
      temp2 : Bool;
      "positive purge on" : Bool;
      temp3 : Bool;
      "close Drain Valves" : Bool;
      RE : Bool;
      RE_1 : Bool;
      RE_2 : Bool;
      "Final Pressure Msg" : Bool;
      Over : Bool;
      "steam purging time actual" : DInt;
      "steam purging done" : Bool;
      "Hot Air Drying" : Bool;
      "Cold Air Drying" : Bool;
      "steam purging time set temp" : DInt;
      "Positive purge over" : Bool;
      temp4 : Bool;
      temp5 : Bool;
      "Startup msg" : Bool;
      "Line valves opening time" : Int;
      "Drain valves opening time" : Int;
      "Actual Set Pulsing Temperature" : Real;
      "Actual Set Pulsing Pressure" : Real;
      "Sterilization Actual Repetition" : Int;
      RE_3 : Bool;
      RE_4 : Bool;
      RE_5 : Bool;
      "Time base air purge" : Bool;
      "Sterilization Start bit" : Bool;
      "Sterilization End bit" : Bool;
      CoolingThresholdTemp : Real;
      StartChillingLine : Bool;
      ChwoValve : Bool;
      PressureReleaseSel : Bool;
      PressureReleaseTime : Int;
      JDBerforeFinalPress : Bool;
      Temp6 : Bool;
      Temp7 : Bool;
      "Sterilization Set RepetitionTemp" : Int;
      ResetSipTimer : Bool;
   END_VAR
   VAR
      "Pulsing Check delay" { S7_SetPoint := 'True'} : "On Delay Timer";
      "SIP HOLD TIMER" { S7_SetPoint := 'True'} : "R_TIMER";
      "Abort temp" { S7_SetPoint := 'True'} : "On Delay Timer";
      "AIR PURGE TIMER" { S7_SetPoint := 'True'} : "R_TIMER";
      "pos purge check" { S7_SetPoint := 'True'} : "On Delay Timer";
      "Steam Purging delay" { S7_SetPoint := 'True'} : "On Delay Timer";
      "Steam purging" { S7_SetPoint := 'True'} : "R_TIMER";
      "Jacket drain" { S7_SetPoint := 'True'} : "On Delay Timer";
      "Delay for Stabilize" { S7_SetPoint := 'True'} : "On Delay Timer";
      PressureReleaseTimer : "R_TIMER";
      OverReset { S7_SetPoint := 'True'} : IEC_TIMER;
      JDBerforeFinalPress_1 : "On Delay Timer";
      IEC_Counter_0_Instance { S7_SetPoint := 'True'} : CTU_INT;
   END_VAR
   VAR_TEMP   // added for the SCL form of the ladder/FBD networks
      _w1 : Bool;
      _w2 : Bool;
      _w3 : Bool;
      _w4 : Bool;
      _w5 : Bool;
      _w6 : Bool;
      _w7 : Bool;
      _w8 : Bool;
      _w9 : Bool;
      _w10 : Bool;
      _w11 : Bool;
   END_VAR
BEGIN

REGION Network 1: Start
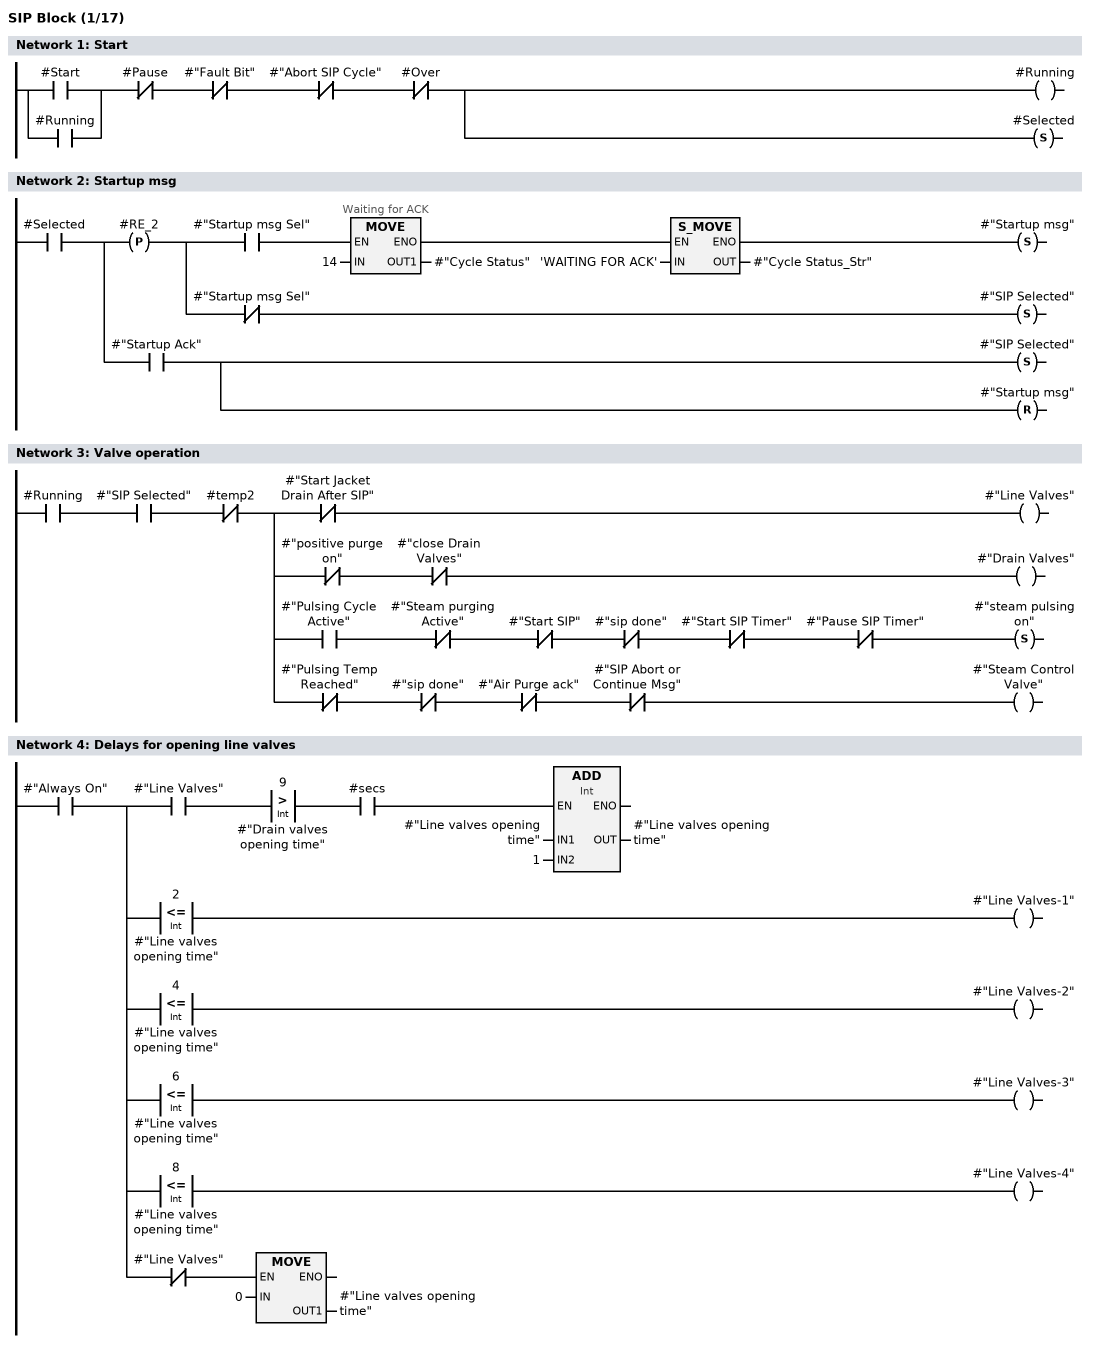
   RUNG wire#powerrail
      Contact( #Start )
      wire#w1
      I_Contact( #Pause )
      I_Contact( #"Fault Bit" )
      I_Contact( #"Abort SIP Cycle" )
      I_Contact( #Over )
      wire#w2
      Coil( #Running )
   END_RUNG
   RUNG wire#powerrail
      Contact( #Running )
   END_RUNG wire#w1
   RUNG wire#w2
      S_Coil( #Selected )
   END_RUNG
   // the same network as SCL:
   #Running := (#Start OR #Running) AND NOT #Pause AND NOT #"Fault Bit" AND NOT #"Abort SIP Cycle" AND NOT #Over;
   IF #Running THEN #Selected := TRUE; END_IF;
END_REGION

REGION Network 2: Startup msg
   RUNG wire#powerrail
      Contact( #Selected )
      wire#w1
      P_Trig( #RE_2 )
      wire#w2
      Contact( #"Startup msg Sel" )
      { S7_GenerateENO := "TRUE" } Move(in := 14, out1 => #"Cycle Status")   // Waiting for ACK
      S_Move(in := 'WAITING FOR ACK', out => #"Cycle Status_Str")
      S_Coil( #"Startup msg" )
   END_RUNG
   RUNG wire#w2
      I_Contact( #"Startup msg Sel" )
      S_Coil( #"SIP Selected" )
   END_RUNG
   RUNG wire#w1
      Contact( #"Startup Ack" )
      wire#w3
      S_Coil( #"SIP Selected" )
   END_RUNG
   RUNG wire#w3
      R_Coil( #"Startup msg" )
   END_RUNG
   // the same network as SCL:
   // ENO of a box is taken as its EN; it also drops when the box reports an error
   #_w1 := #Selected AND NOT #RE_2;   // rising edge
   #RE_2 := #Selected;
   IF #_w1 AND #"Startup msg Sel" THEN
       #"Cycle Status" := 14;   // Waiting for ACK
       #"Cycle Status_Str" := 'WAITING FOR ACK';
       #"Startup msg" := TRUE;
   END_IF;
   IF #_w1 AND NOT #"Startup msg Sel" THEN #"SIP Selected" := TRUE; END_IF;
   IF #Selected AND #"Startup Ack" THEN
       #"SIP Selected" := TRUE;
       #"Startup msg" := FALSE;
   END_IF;
END_REGION

REGION Network 3: Valve operation
   RUNG wire#powerrail
      Contact( #Running )
      Contact( #"SIP Selected" )
      I_Contact( #temp2 )
      wire#w1
      I_Contact( #"Start Jacket Drain After SIP" )
      Coil( #"Line Valves" )
   END_RUNG
   RUNG wire#w1
      I_Contact( #"positive purge on" )
      I_Contact( #"close Drain Valves" )
      Coil( #"Drain Valves" )
   END_RUNG
   RUNG wire#w1
      Contact( #"Pulsing Cycle Active" )
      I_Contact( #"Steam purging Active" )
      I_Contact( #"Start SIP" )
      I_Contact( #"sip done" )
      I_Contact( #"Start SIP Timer" )
      I_Contact( #"Pause SIP Timer" )
      S_Coil( #"steam pulsing on" )
   END_RUNG
   RUNG wire#w1
      I_Contact( #"Pulsing Temp Reached" )
      I_Contact( #"sip done" )
      I_Contact( #"Air Purge ack" )
      I_Contact( #"SIP Abort or Continue Msg" )
      Coil( #"Steam Control Valve" )
   END_RUNG
   // the same network as SCL:
   #_w1 := #Running AND #"SIP Selected" AND NOT #temp2;
   #"Line Valves" := #_w1 AND NOT #"Start Jacket Drain After SIP";
   #"Drain Valves" := #_w1 AND NOT #"positive purge on" AND NOT #"close Drain Valves";
   IF #_w1 AND #"Pulsing Cycle Active" AND NOT #"Steam purging Active" AND NOT #"Start SIP" AND NOT #"sip done" AND NOT #"Start SIP Timer" AND NOT #"Pause SIP Timer" THEN
       #"steam pulsing on" := TRUE;
   END_IF;
   #"Steam Control Valve" := #_w1 AND NOT #"Pulsing Temp Reached" AND NOT #"sip done" AND NOT #"Air Purge ack" AND NOT #"SIP Abort or Continue Msg";
END_REGION

REGION Network 4: Delays for opening line valves
   RUNG wire#powerrail
      Contact( #"Always On" )
      wire#w1
      Contact( #"Line Valves" )
      { S7_Templates := "SrcType := Int" } GT_Contact(in1 := 9, in2 := #"Drain valves opening time")
      Contact( #secs )
      { S7_Templates := "SrcType := Int"; S7_GenerateENO := "TRUE" } Add(in1 := #"Line valves opening time", in2 := 1, out => #"Line valves opening time")
   END_RUNG
   RUNG wire#w1
      { S7_Templates := "SrcType := Int" } LE_Contact(in1 := 2, in2 := #"Line valves opening time")
      Coil( #"Line Valves-1" )
   END_RUNG
   RUNG wire#w1
      { S7_Templates := "SrcType := Int" } LE_Contact(in1 := 4, in2 := #"Line valves opening time")
      Coil( #"Line Valves-2" )
   END_RUNG
   RUNG wire#w1
      { S7_Templates := "SrcType := Int" } LE_Contact(in1 := 6, in2 := #"Line valves opening time")
      Coil( #"Line Valves-3" )
   END_RUNG
   RUNG wire#w1
      { S7_Templates := "SrcType := Int" } LE_Contact(in1 := 8, in2 := #"Line valves opening time")
      Coil( #"Line Valves-4" )
   END_RUNG
   RUNG wire#w1
      I_Contact( #"Line Valves" )
      { S7_GenerateENO := "TRUE" } Move(in := 0, out1 => #"Line valves opening time")
   END_RUNG
   // the same network as SCL:
   IF #"Always On" AND #"Line Valves" AND (9 > #"Drain valves opening time") AND #secs THEN
       #"Line valves opening time" := #"Line valves opening time" + 1;
   END_IF;
   #"Line Valves-1" := #"Always On" AND (2 <= #"Line valves opening time");
   #"Line Valves-2" := #"Always On" AND (4 <= #"Line valves opening time");
   #"Line Valves-3" := #"Always On" AND (6 <= #"Line valves opening time");
   #"Line Valves-4" := #"Always On" AND (8 <= #"Line valves opening time");
   IF #"Always On" AND NOT #"Line Valves" THEN #"Line valves opening time" := 0; END_IF;
END_REGION

REGION Network 5: Delays for opening drain valves
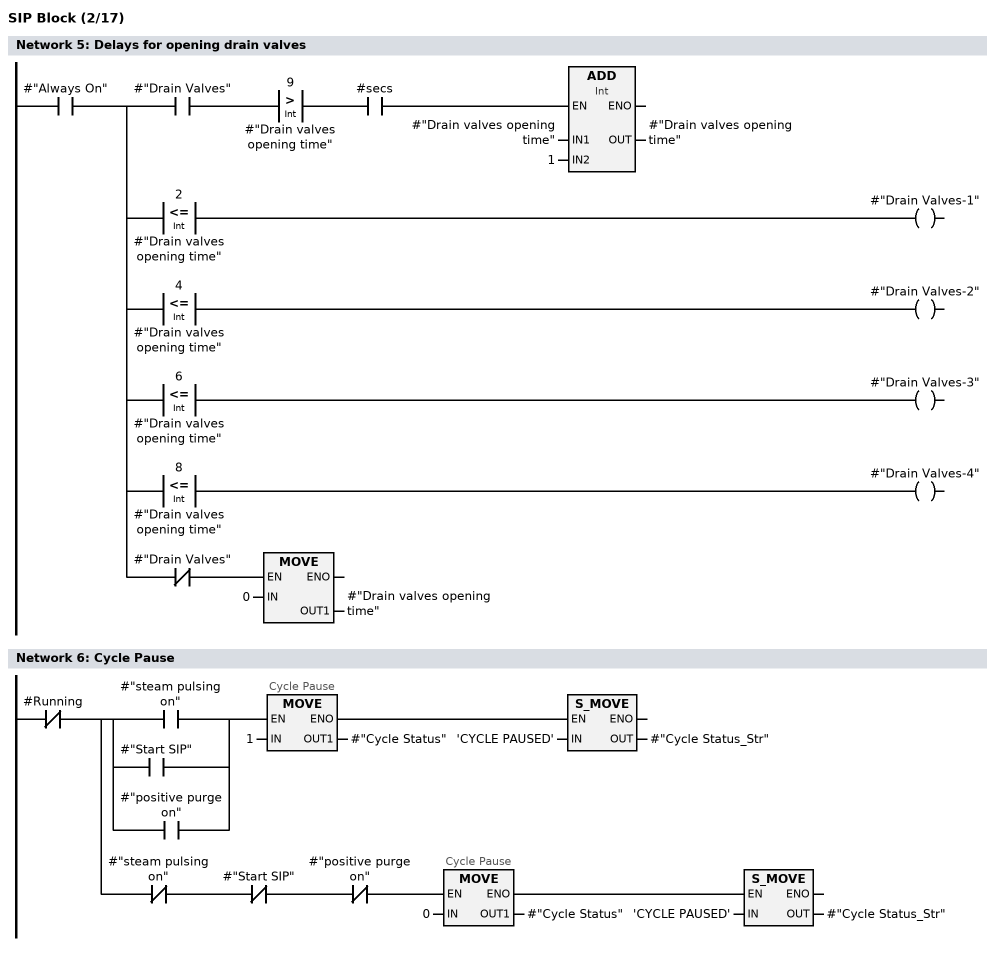
   RUNG wire#powerrail
      Contact( #"Always On" )
      wire#w1
      Contact( #"Drain Valves" )
      { S7_Templates := "SrcType := Int" } GT_Contact(in1 := 9, in2 := #"Drain valves opening time")
      Contact( #secs )
      { S7_Templates := "SrcType := Int"; S7_GenerateENO := "TRUE" } Add(in1 := #"Drain valves opening time", in2 := 1, out => #"Drain valves opening time")
   END_RUNG
   RUNG wire#w1
      { S7_Templates := "SrcType := Int" } LE_Contact(in1 := 2, in2 := #"Drain valves opening time")
      Coil( #"Drain Valves-1" )
   END_RUNG
   RUNG wire#w1
      { S7_Templates := "SrcType := Int" } LE_Contact(in1 := 4, in2 := #"Drain valves opening time")
      Coil( #"Drain Valves-2" )
   END_RUNG
   RUNG wire#w1
      { S7_Templates := "SrcType := Int" } LE_Contact(in1 := 6, in2 := #"Drain valves opening time")
      Coil( #"Drain Valves-3" )
   END_RUNG
   RUNG wire#w1
      { S7_Templates := "SrcType := Int" } LE_Contact(in1 := 8, in2 := #"Drain valves opening time")
      Coil( #"Drain Valves-4" )
   END_RUNG
   RUNG wire#w1
      I_Contact( #"Drain Valves" )
      { S7_GenerateENO := "TRUE" } Move(in := 0, out1 => #"Drain valves opening time")
   END_RUNG
   // the same network as SCL:
   IF #"Always On" AND #"Drain Valves" AND (9 > #"Drain valves opening time") AND #secs THEN
       #"Drain valves opening time" := #"Drain valves opening time" + 1;
   END_IF;
   #"Drain Valves-1" := #"Always On" AND (2 <= #"Drain valves opening time");
   #"Drain Valves-2" := #"Always On" AND (4 <= #"Drain valves opening time");
   #"Drain Valves-3" := #"Always On" AND (6 <= #"Drain valves opening time");
   #"Drain Valves-4" := #"Always On" AND (8 <= #"Drain valves opening time");
   IF #"Always On" AND NOT #"Drain Valves" THEN #"Drain valves opening time" := 0; END_IF;
END_REGION

REGION Network 6: Cycle Pause
   RUNG wire#powerrail
      I_Contact( #Running )
      wire#w1
      Contact( #"steam pulsing on" )
      wire#w2
      { S7_GenerateENO := "TRUE" } Move(in := 1, out1 => #"Cycle Status")   // Cycle Pause
      S_Move(in := 'CYCLE PAUSED', out => #"Cycle Status_Str")
   END_RUNG
   RUNG wire#w1
      Contact( #"Start SIP" )
   END_RUNG wire#w2
   RUNG wire#w1
      Contact( #"positive purge on" )
   END_RUNG wire#w2
   RUNG wire#w1
      I_Contact( #"steam pulsing on" )
      I_Contact( #"Start SIP" )
      I_Contact( #"positive purge on" )
      { S7_GenerateENO := "TRUE" } Move(in := 0, out1 => #"Cycle Status")   // Cycle Pause
      S_Move(in := 'CYCLE PAUSED', out => #"Cycle Status_Str")
   END_RUNG
   // the same network as SCL:
   // ENO of a box is taken as its EN; it also drops when the box reports an error
   IF NOT #Running AND (#"steam pulsing on" OR #"Start SIP" OR #"positive purge on") THEN
       #"Cycle Status" := 1;   // Cycle Pause
       #"Cycle Status_Str" := 'CYCLE PAUSED';
   END_IF;
   IF NOT #Running AND NOT #"steam pulsing on" AND NOT #"Start SIP" AND NOT #"positive purge on" THEN
       #"Cycle Status" := 0;   // Cycle Pause
       #"Cycle Status_Str" := 'CYCLE PAUSED';
   END_IF;
END_REGION

REGION Network 7: Steam purging
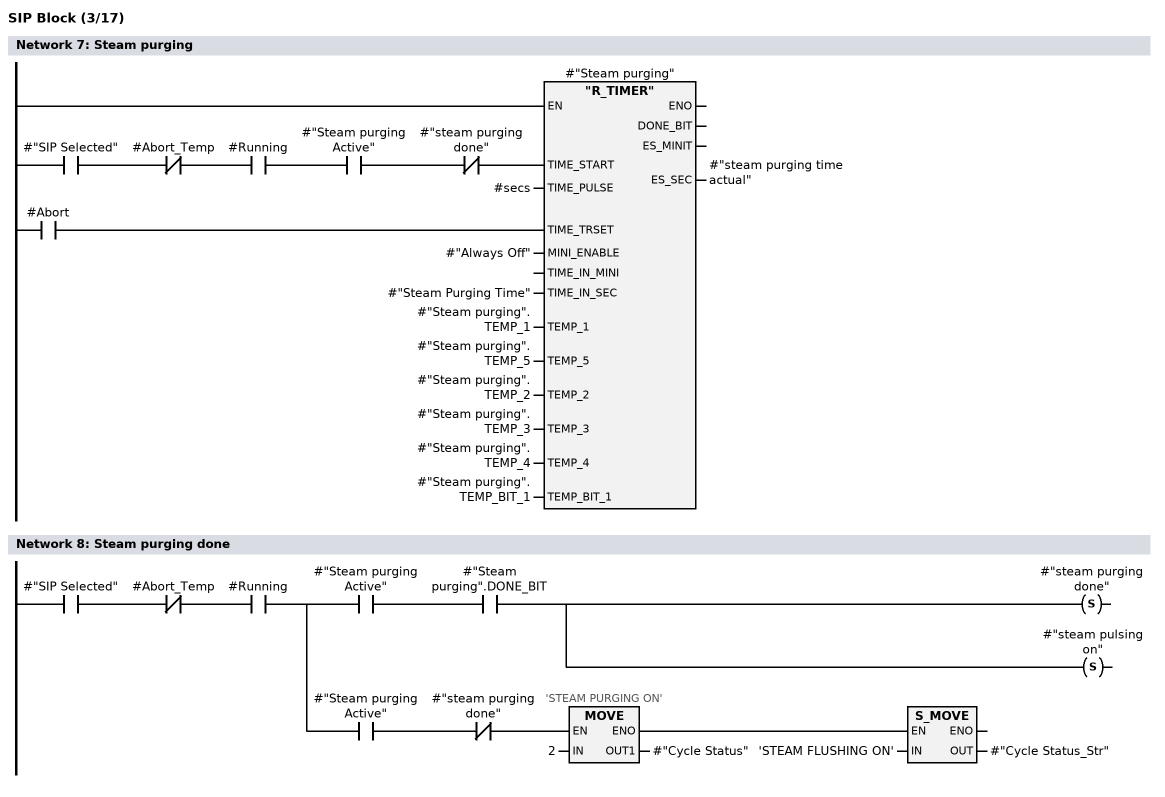
   RUNG wire#powerrail
      #"Steam purging"(TIME_START := wire#w1, TIME_TRSET := wire#w2, TIME_PULSE := #secs, MINI_ENABLE := #"Always Off", TIME_IN_MINI :=, TIME_IN_SEC := #"Steam Purging Time", TEMP_1 := #"Steam purging".TEMP_1, TEMP_5 := #"Steam purging".TEMP_5, TEMP_2 := #"Steam purging".TEMP_2, TEMP_3 := #"Steam purging".TEMP_3, TEMP_4 := #"Steam purging".TEMP_4, TEMP_BIT_1 := #"Steam purging".TEMP_BIT_1, DONE_BIT =>, ES_MINIT =>, ES_SEC => #"steam purging time actual")
   END_RUNG
   RUNG wire#powerrail
      Contact( #"SIP Selected" )
      I_Contact( #Abort_Temp )
      Contact( #Running )
      Contact( #"Steam purging Active" )
      I_Contact( #"steam purging done" )
   END_RUNG wire#w1
   RUNG wire#powerrail
      Contact( #Abort )
   END_RUNG wire#w2
   // the same network as SCL:
   #"Steam purging"(TIME_START := #"SIP Selected" AND NOT #Abort_Temp AND #Running AND #"Steam purging Active" AND NOT #"steam purging done",   // "R_TIMER"
                    TIME_PULSE := #secs,
                    TIME_TRSET := #Abort,
                    MINI_ENABLE := #"Always Off",
                    TIME_IN_SEC := #"Steam Purging Time",
                    TEMP_1 := #"Steam purging".TEMP_1,
                    TEMP_5 := #"Steam purging".TEMP_5,
                    TEMP_2 := #"Steam purging".TEMP_2,
                    TEMP_3 := #"Steam purging".TEMP_3,
                    TEMP_4 := #"Steam purging".TEMP_4,
                    TEMP_BIT_1 := #"Steam purging".TEMP_BIT_1,
                    ES_SEC => #"steam purging time actual");
END_REGION

REGION Network 8: Steam purging done
   RUNG wire#powerrail
      Contact( #"SIP Selected" )
      I_Contact( #Abort_Temp )
      Contact( #Running )
      wire#w1
      Contact( #"Steam purging Active" )
      Contact( #"Steam purging".DONE_BIT )
      wire#w2
      S_Coil( #"steam purging done" )
   END_RUNG
   RUNG wire#w2
      S_Coil( #"steam pulsing on" )
   END_RUNG
   RUNG wire#w1
      Contact( #"Steam purging Active" )
      I_Contact( #"steam purging done" )
      { S7_GenerateENO := "TRUE" } Move(in := 2, out1 => #"Cycle Status")   // 'STEAM PURGING ON'
      S_Move(in := 'STEAM FLUSHING ON', out => #"Cycle Status_Str")
   END_RUNG
   // the same network as SCL:
   // ENO of a box is taken as its EN; it also drops when the box reports an error
   #_w1 := #"SIP Selected" AND NOT #Abort_Temp AND #Running;
   IF #_w1 AND #"Steam purging Active" AND #"Steam purging".DONE_BIT THEN
       #"steam purging done" := TRUE;
       #"steam pulsing on" := TRUE;
   END_IF;
   IF #_w1 AND #"Steam purging Active" AND NOT #"steam purging done" THEN
       #"Cycle Status" := 2;   // 'STEAM PURGING ON'
       #"Cycle Status_Str" := 'STEAM FLUSHING ON';
   END_IF;
END_REGION

REGION Network 9: #"Pulsing Temp Reached"
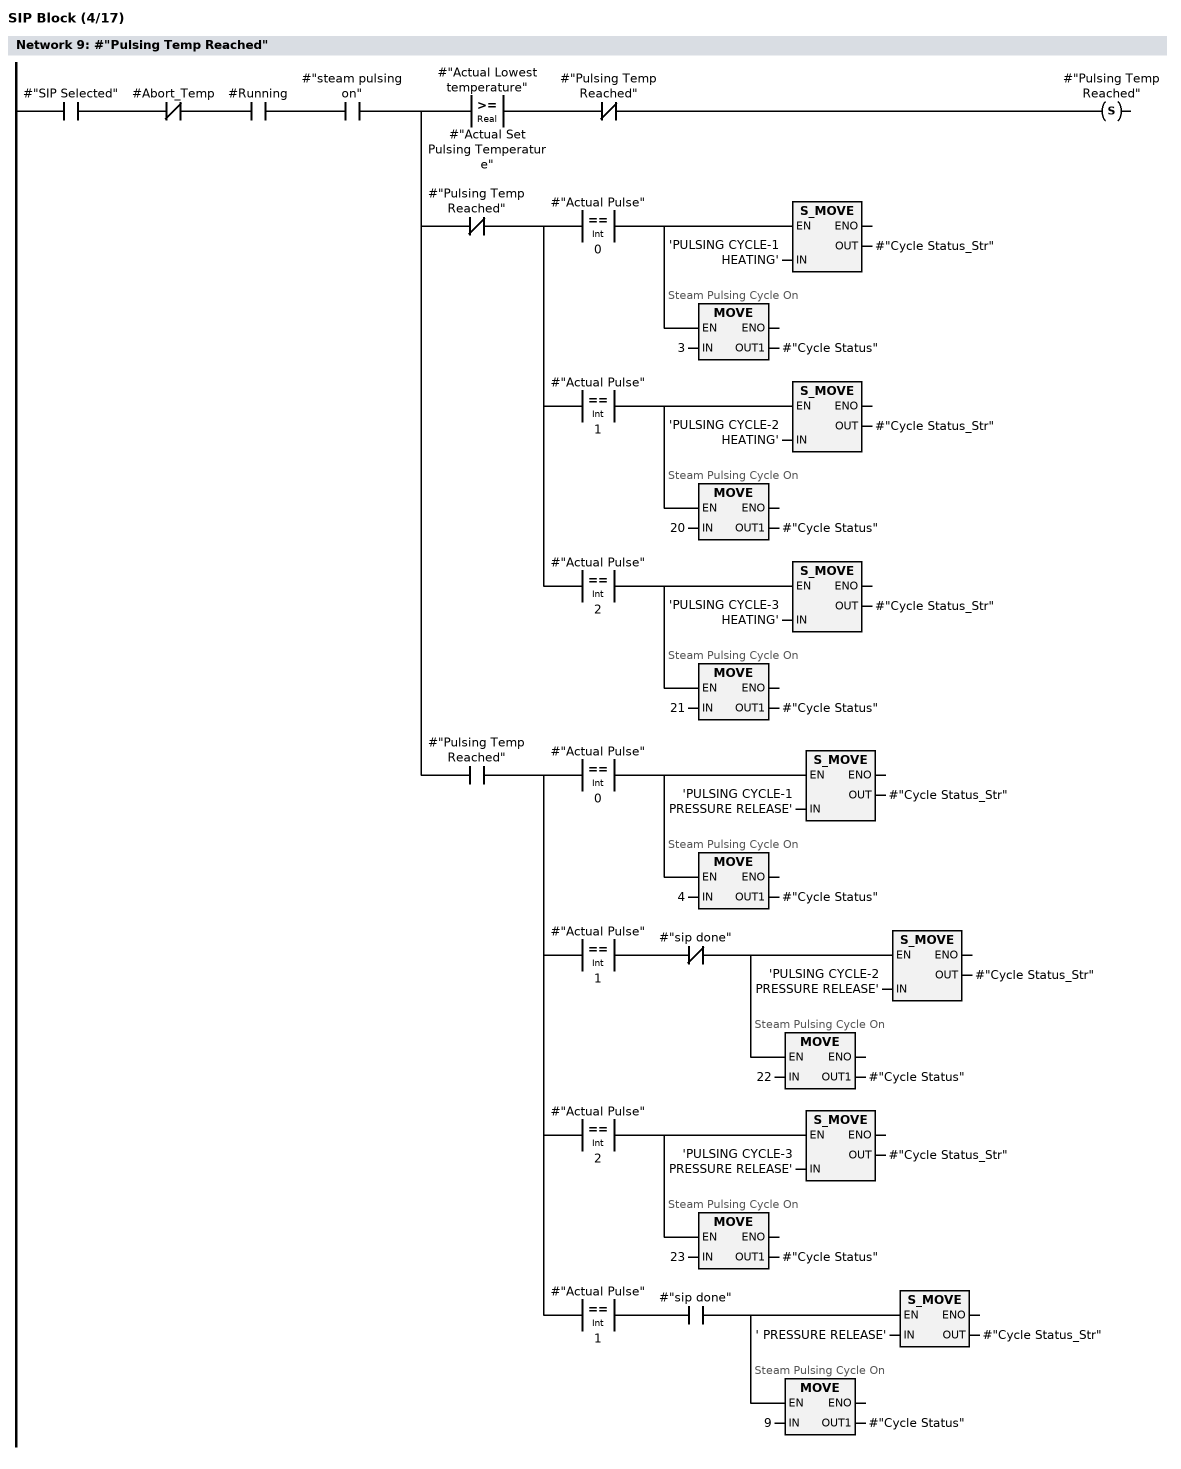
   RUNG wire#powerrail
      Contact( #"SIP Selected" )
      I_Contact( #Abort_Temp )
      Contact( #Running )
      Contact( #"steam pulsing on" )
      wire#w1
      { S7_Templates := "SrcType := Real" } GE_Contact(in1 := #"Actual Lowest temperature", in2 := #"Actual Set Pulsing Temperature")
      I_Contact( #"Pulsing Temp Reached" )
      S_Coil( #"Pulsing Temp Reached" )
   END_RUNG
   RUNG wire#w1
      I_Contact( #"Pulsing Temp Reached" )
      wire#w2
      { S7_Templates := "SrcType := Int" } EQ_Contact(in1 := #"Actual Pulse", in2 := 0)
      wire#w3
      S_Move(in := 'PULSING CYCLE-1 HEATING', out => #"Cycle Status_Str")
   END_RUNG
   RUNG wire#w3
      { S7_GenerateENO := "TRUE" } Move(in := 3, out1 => #"Cycle Status")   // Steam Pulsing Cycle On
   END_RUNG
   RUNG wire#w2
      { S7_Templates := "SrcType := Int" } EQ_Contact(in1 := #"Actual Pulse", in2 := 1)
      wire#w4
      S_Move(in := 'PULSING CYCLE-2 HEATING', out => #"Cycle Status_Str")
   END_RUNG
   RUNG wire#w4
      { S7_GenerateENO := "TRUE" } Move(in := 20, out1 => #"Cycle Status")   // Steam Pulsing Cycle On
   END_RUNG
   RUNG wire#w2
      { S7_Templates := "SrcType := Int" } EQ_Contact(in1 := #"Actual Pulse", in2 := 2)
      wire#w5
      S_Move(in := 'PULSING CYCLE-3 HEATING', out => #"Cycle Status_Str")
   END_RUNG
   RUNG wire#w5
      { S7_GenerateENO := "TRUE" } Move(in := 21, out1 => #"Cycle Status")   // Steam Pulsing Cycle On
   END_RUNG
   RUNG wire#w1
      Contact( #"Pulsing Temp Reached" )
      wire#w6
      { S7_Templates := "SrcType := Int" } EQ_Contact(in1 := #"Actual Pulse", in2 := 0)
      wire#w7
      S_Move(in := 'PULSING CYCLE-1 PRESSURE RELEASE', out => #"Cycle Status_Str")
   END_RUNG
   RUNG wire#w7
      { S7_GenerateENO := "TRUE" } Move(in := 4, out1 => #"Cycle Status")   // Steam Pulsing Cycle On
   END_RUNG
   RUNG wire#w6
      { S7_Templates := "SrcType := Int" } EQ_Contact(in1 := #"Actual Pulse", in2 := 1)
      I_Contact( #"sip done" )
      wire#w8
      S_Move(in := 'PULSING CYCLE-2 PRESSURE RELEASE', out => #"Cycle Status_Str")
   END_RUNG
   RUNG wire#w8
      { S7_GenerateENO := "TRUE" } Move(in := 22, out1 => #"Cycle Status")   // Steam Pulsing Cycle On
   END_RUNG
   RUNG wire#w6
      { S7_Templates := "SrcType := Int" } EQ_Contact(in1 := #"Actual Pulse", in2 := 2)
      wire#w9
      S_Move(in := 'PULSING CYCLE-3 PRESSURE RELEASE', out => #"Cycle Status_Str")
   END_RUNG
   RUNG wire#w9
      { S7_GenerateENO := "TRUE" } Move(in := 23, out1 => #"Cycle Status")   // Steam Pulsing Cycle On
   END_RUNG
   RUNG wire#w6
      { S7_Templates := "SrcType := Int" } EQ_Contact(in1 := #"Actual Pulse", in2 := 1)
      Contact( #"sip done" )
      wire#w10
      S_Move(in := ' PRESSURE RELEASE', out => #"Cycle Status_Str")
   END_RUNG
   RUNG wire#w10
      { S7_GenerateENO := "TRUE" } Move(in := 9, out1 => #"Cycle Status")   // Steam Pulsing Cycle On
   END_RUNG
   // the same network as SCL:
   #_w1 := #"SIP Selected" AND NOT #Abort_Temp AND #Running AND #"steam pulsing on";
   IF #_w1 AND (#"Actual Lowest temperature" >= #"Actual Set Pulsing Temperature") AND NOT #"Pulsing Temp Reached" THEN
       #"Pulsing Temp Reached" := TRUE;
   END_IF;
   #_w2 := #_w1 AND NOT #"Pulsing Temp Reached";
   IF #_w2 AND (#"Actual Pulse" = 0) THEN
       #"Cycle Status_Str" := 'PULSING CYCLE-1 HEATING';
       #"Cycle Status" := 3;   // Steam Pulsing Cycle On
   END_IF;
   IF #_w2 AND (#"Actual Pulse" = 1) THEN
       #"Cycle Status_Str" := 'PULSING CYCLE-2 HEATING';
       #"Cycle Status" := 20;   // Steam Pulsing Cycle On
   END_IF;
   IF #_w2 AND (#"Actual Pulse" = 2) THEN
       #"Cycle Status_Str" := 'PULSING CYCLE-3 HEATING';
       #"Cycle Status" := 21;   // Steam Pulsing Cycle On
   END_IF;
   #_w3 := #_w1 AND #"Pulsing Temp Reached";
   IF #_w3 AND (#"Actual Pulse" = 0) THEN
       #"Cycle Status_Str" := 'PULSING CYCLE-1 PRESSURE RELEASE';
       #"Cycle Status" := 4;   // Steam Pulsing Cycle On
   END_IF;
   IF #_w3 AND (#"Actual Pulse" = 1) AND NOT #"sip done" THEN
       #"Cycle Status_Str" := 'PULSING CYCLE-2 PRESSURE RELEASE';
       #"Cycle Status" := 22;   // Steam Pulsing Cycle On
   END_IF;
   IF #_w3 AND (#"Actual Pulse" = 2) THEN
       #"Cycle Status_Str" := 'PULSING CYCLE-3 PRESSURE RELEASE';
       #"Cycle Status" := 23;   // Steam Pulsing Cycle On
   END_IF;
   IF #_w3 AND (#"Actual Pulse" = 1) AND #"sip done" THEN
       #"Cycle Status_Str" := ' PRESSURE RELEASE';
       #"Cycle Status" := 9;   // Steam Pulsing Cycle On
   END_IF;
END_REGION

